LIN {X 0,Y 298.413,Z 394.313,A -85,B 0,C 180,E1 -16229.642,E2 -16229.642} C_VEL
LIN {X 0,Y 298.389,Z 394.317,A -85,B 0,C 180,E1 -16232.801,E2 -16232.801} C_VEL
LIN {X 0,Y 298.456,Z 394.307,A -85,B 0,C 180,E1 -16236.814,E2 -16236.814} C_VEL
LIN {X 0,Y 298.404,Z 394.314,A -85,B 0,C 180,E1 -16241.095,E2 -16241.095} C_VEL
LIN {X 0,Y 298.418,Z 394.313,A -85,B 0,C 180,E1 -16243.11,E2 -16243.11} C_VEL
LIN {X 0,Y 298.396,Z 394.317,A -85,B 0,C 180,E1 -16246.922,E2 -16246.922} C_VEL
LIN {X 0,Y 298.398,Z 394.314,A -85,B 0,C 180,E1 -16251.008,E2 -16251.008} C_VEL
LIN {X 0,Y 298.421,Z 394.313,A -85,B 0,C 180,E1 -16254.764,E2 -16254.764} C_VEL
LIN {X 0,Y 298.43,Z 394.322,A -85,B 0,C 180,E1 -16255.234,E2 -16255.234} C_VEL
LIN {X 0,Y 298.861,Z 396.048,A -85,B 0,C 180,E1 -16255.643,E2 -16255.643} C_VEL
LIN {X 0,Y 302.324,Z 402.19,A -85,B 0,C 180,E1 -16257.395,E2 -16257.395} C_VEL
LIN {X 0,Y 303.861,Z 406.66,A -85,B 0,C 180,E1 -16258.271,E2 -16258.271} C_VEL
LIN {X 0,Y 306.901,Z 413.206,A -85,B 0,C 180,E1 -16259.176,E2 -16259.176} C_VEL
LIN {X 0,Y 310.226,Z 420.843,A -85,B 0,C 180,E1 -16260.12,E2 -16260.12} C_VEL
LIN {X 0,Y 313.351,Z 428.982,A -85,B 0,C 180,E1 -16261.011,E2 -16261.011} C_VEL
LIN {X 0,Y 315.702,Z 443.344,A -85,B 0,C 180,E1 -16261.99,E2 -16261.99} C_VEL
LIN {X 0,Y 317.187,Z 456.396,A -85,B 0,C 180,E1 -16262.756,E2 -16262.756} C_VEL
LIN {X 0,Y 317.42,Z 461.154,A -85,B 0,C 180,E1 -16262.981,E2 -16262.981} C_VEL
LIN {X 0,Y 313.679,Z 525.311,A -85,B 0,C 180,E1 -16265.029,E2 -16265.029} C_VEL
LIN {X 0,Y 312.276,Z 538.46,A -85,B 0,C 180,E1 -16265.663,E2 -16265.663} C_VEL
LIN {X 0,Y 310.663,Z 550.678,A -85,B 0,C 180,E1 -16266.504,E2 -16266.504} C_VEL
LIN {X 0,Y 308.807,Z 562.616,A -85,B 0,C 180,E1 -16267.594,E2 -16267.594} C_VEL
LIN {X 0,Y 306.824,Z 573.531,A -85,B 0,C 180,E1 -16268.855,E2 -16268.855} C_VEL
LIN {X 0,Y 304.681,Z 584.454,A -85,B 0,C 180,E1 -16270.462,E2 -16270.462} C_VEL
LIN {X 0,Y 302.875,Z 593.194,A -85,B 0,C 180,E1 -16272.06,E2 -16272.06} C_VEL
LIN {X 0,Y 301.068,Z 602.117,A -85,B 0,C 180,E1 -16274.082,E2 -16274.082} C_VEL
LIN {X 0,Y 299.516,Z 609.166,A -85,B 0,C 180,E1 -16276.085,E2 -16276.085} C_VEL
LIN {X 0,Y 298.089,Z 615.668,A -85,B 0,C 180,E1 -16278.441,E2 -16278.441} C_VEL
LIN {X 0,Y 297.32,Z 619.91,A -85,B 0,C 180,E1 -16280.478,E2 -16280.478} C_VEL
LIN {X 0,Y 296.96,Z 622.117,A -85,B 0,C 180,E1 -16281.838,E2 -16281.838} C_VEL
LIN {X 0,Y 296.586,Z 625.088,A -85,B 0,C 180,E1 -16284.412,E2 -16284.412} C_VEL
LIN {X 0,Y 296.494,Z 627.829,A -85,B 0,C 180,E1 -16288.644,E2 -16288.644} C_VEL
LIN {X 0,Y 296.518,Z 628.283,A -85,B 0,C 180,E1 -16290.002,E2 -16290.002} C_VEL
LIN {X 0,Y 296.485,Z 628.313,A -85,B 0,C 180,E1 -16291.36,E2 -16291.36} C_VEL
LIN {X 0,Y 296.527,Z 627.952,A -85,B 0,C 180,E1 -16292.719,E2 -16292.719} C_VEL
LIN {X 0,Y 296.493,Z 627.197,A -85,B 0,C 180,E1 -16294.08,E2 -16294.08} C_VEL
LIN {X 0,Y 296.547,Z 625.934,A -85,B 0,C 180,E1 -16295.51,E2 -16295.51} C_VEL
LIN {X 0,Y 296.948,Z 622.356,A -85,B 0,C 180,E1 -16298.166,E2 -16298.166} C_VEL
LIN {X 0,Y 297.479,Z 618.423,A -85,B 0,C 180,E1 -16300.208,E2 -16300.208} C_VEL
LIN {X 0,Y 298.337,Z 613.363,A -85,B 0,C 180,E1 -16302.242,E2 -16302.242} C_VEL
LIN {X 0,Y 299.641,Z 607.023,A -85,B 0,C 180,E1 -16304.259,E2 -16304.259} C_VEL
LIN {X 0,Y 301.128,Z 599.116,A -85,B 0,C 180,E1 -16306.266,E2 -16306.266} C_VEL
LIN {X 0,Y 302.907,Z 589.288,A -85,B 0,C 180,E1 -16308.255,E2 -16308.255} C_VEL
LIN {X 0,Y 304.715,Z 579.147,A -85,B 0,C 180,E1 -16309.89,E2 -16309.89} C_VEL
LIN {X 0,Y 306.713,Z 567.717,A -85,B 0,C 180,E1 -16311.333,E2 -16311.333} C_VEL
LIN {X 0,Y 308.342,Z 556.565,A -85,B 0,C 180,E1 -16312.446,E2 -16312.446} C_VEL
LIN {X 0,Y 309.823,Z 544.144,A -85,B 0,C 180,E1 -16313.39,E2 -16313.39} C_VEL
LIN {X 0,Y 311.118,Z 531.155,A -85,B 0,C 180,E1 -16314.08,E2 -16314.08} C_VEL
LIN {X 0,Y 311.871,Z 518.085,A -85,B 0,C 180,E1 -16314.534,E2 -16314.534} C_VEL
LIN {X 0,Y 313.809,Z 459.058,A -85,B 0,C 180,E1 -16316.022,E2 -16316.022} C_VEL
LIN {X 0,Y 310.871,Z 439.691,A -85,B 0,C 180,E1 -16316.91,E2 -16316.91} C_VEL
LIN {X 0,Y 308.062,Z 426.174,A -85,B 0,C 180,E1 -16317.642,E2 -16317.642} C_VEL
LIN {X 0,Y 303.315,Z 415.098,A -85,B 0,C 180,E1 -16318.585,E2 -16318.585} C_VEL
LIN {X 0,Y 301.215,Z 405.403,A -85,B 0,C 180,E1 -16322.062,E2 -16322.062} C_VEL
LIN {X 0,Y 299.211,Z 397.209,A -85,B 0,C 180,E1 -16325.239,E2 -16325.239} C_VEL
LIN {X 0,Y 298.473,Z 394.309,A -85,B 0,C 180,E1 -16326.437,E2 -16326.437} C_VEL
LIN {X 0,Y 298.414,Z 394.321,A -85,B 0,C 180,E1 -16329.487,E2 -16329.487} C_VEL
LIN {X 0,Y 298.404,Z 394.318,A -85,B 0,C 180,E1 -16333.104,E2 -16333.104} C_VEL
LIN {X 0,Y 298.408,Z 394.312,A -85,B 0,C 180,E1 -16336.922,E2 -16336.922} C_VEL
LIN {X 0,Y 298.41,Z 394.314,A -85,B 0,C 180,E1 -16341.007,E2 -16341.007} C_VEL
LIN {X 0,Y 298.425,Z 394.31,A -85,B 0,C 180,E1 -16343.931,E2 -16343.931} C_VEL
LIN {X 0,Y 298.4,Z 394.314,A -85,B 0,C 180,E1 -16347.985,E2 -16347.985} C_VEL
LIN {X 0,Y 298.463,Z 394.306,A -85,B 0,C 180,E1 -16351.904,E2 -16351.904} C_VEL
LIN {X 0,Y 298.49,Z 394.305,A -85,B 0,C 180,E1 -16354.924,E2 -16354.924} C_VEL
LIN {X 0,Y 298.457,Z 394.308,A -85,B 0,C 180,E1 -16359.316,E2 -16359.316} C_VEL
LIN {X 0,Y 298.545,Z 394.289,A -85,B 0,C 180,E1 -16362.18,E2 -16362.18} C_VEL
LIN {X 0,Y 298.6,Z 394.28,A -85,B 0,C 180,E1 -16364.995,E2 -16364.995} C_VEL
LIN {X 0,Y 298.6,Z 394.28,A -85,B 0,C 180,E1 -16369.147,E2 -16369.147} C_VEL
LIN {X 0,Y 298.766,Z 394.271,A -85,B 0,C 180,E1 -16371.886,E2 -16371.886} C_VEL
LIN {X 0,Y 298.667,Z 394.28,A -85,B 0,C 180,E1 -16374.599,E2 -16374.599} C_VEL
LIN {X 0,Y 298.929,Z 394.25,A -85,B 0,C 180,E1 -16378.653,E2 -16378.653} C_VEL
LIN {X 0,Y 298.929,Z 394.245,A -85,B 0,C 180,E1 -16381.347,E2 -16381.347} C_VEL
LIN {X 0,Y 298.805,Z 394.26,A -85,B 0,C 180,E1 -16386.754,E2 -16386.754} C_VEL
LIN {X 0,Y 298.688,Z 394.277,A -85,B 0,C 180,E1 -16389.48,E2 -16389.48} C_VEL
LIN {X 0,Y 298.559,Z 394.295,A -85,B 0,C 180,E1 -16393.615,E2 -16393.615} C_VEL
LIN {X 0,Y 298.556,Z 394.296,A -85,B 0,C 180,E1 -16396.408,E2 -16396.408} C_VEL
LIN {X 0,Y 298.556,Z 394.478,A -85,B 0,C 180,E1 -16399.762,E2 -16399.762} C_VEL
LIN {X 0,Y 300.424,Z 402.299,A -85,B 0,C 180,E1 -16403.115,E2 -16403.115} C_VEL
LIN {X 0,Y 308.076,Z 417.875,A -85,B 0,C 180,E1 -16404.576,E2 -16404.576} C_VEL
LIN {X 0,Y 313.726,Z 431.385,A -85,B 0,C 180,E1 -16405.635,E2 -16405.635} C_VEL
LIN {X 0,Y 314.519,Z 435.202,A -85,B 0,C 180,E1 -16405.832,E2 -16405.832} C_VEL
LIN {X 0,Y 311.916,Z 509.359,A -85,B 0,C 180,E1 -16407.731,E2 -16407.731} C_VEL
LIN {X 0,Y 311.021,Z 522.182,A -85,B 0,C 180,E1 -16408.298,E2 -16408.298} C_VEL
LIN {X 0,Y 309.823,Z 534.58,A -85,B 0,C 180,E1 -16409.097,E2 -16409.097} C_VEL
LIN {X 0,Y 308.255,Z 547.18,A -85,B 0,C 180,E1 -16410.211,E2 -16410.211} C_VEL
LIN {X 0,Y 306.574,Z 558.665,A -85,B 0,C 180,E1 -16411.537,E2 -16411.537} C_VEL
LIN {X 0,Y 304.885,Z 568.72,A -85,B 0,C 180,E1 -16412.997,E2 -16412.997} C_VEL
LIN {X 0,Y 303.175,Z 577.721,A -85,B 0,C 180,E1 -16414.618,E2 -16414.618} C_VEL
LIN {X 0,Y 301.474,Z 586.009,A -85,B 0,C 180,E1 -16416.458,E2 -16416.458} C_VEL
LIN {X 0,Y 300.068,Z 592.824,A -85,B 0,C 180,E1 -16418.328,E2 -16418.328} C_VEL
LIN {X 0,Y 298.765,Z 599.542,A -85,B 0,C 180,E1 -16420.671,E2 -16420.671} C_VEL
LIN {X 0,Y 297.704,Z 604.913,A -85,B 0,C 180,E1 -16423.206,E2 -16423.206} C_VEL
LIN {X 0,Y 297.085,Z 607.992,A -85,B 0,C 180,E1 -16425.211,E2 -16425.211} C_VEL
LIN {X 0,Y 296.595,Z 610.168,A -85,B 0,C 180,E1 -16427.271,E2 -16427.271} C_VEL
LIN {X 0,Y 296.321,Z 611.406,A -85,B 0,C 180,E1 -16429.373,E2 -16429.373} C_VEL
LIN {X 0,Y 296.196,Z 611.621,A -85,B 0,C 180,E1 -16431.907,E2 -16431.907} C_VEL
LIN {X 0,Y 296.212,Z 610.875,A -85,B 0,C 180,E1 -16433.775,E2 -16433.775} C_VEL
LIN {X 0,Y 296.464,Z 608.905,A -85,B 0,C 180,E1 -16436.07,E2 -16436.07} C_VEL
LIN {X 0,Y 296.925,Z 605.306,A -85,B 0,C 180,E1 -16438.617,E2 -16438.617} C_VEL
LIN {X 0,Y 297.467,Z 600.516,A -85,B 0,C 180,E1 -16440.947,E2 -16440.947} C_VEL
LIN {X 0,Y 298.229,Z 594.935,A -85,B 0,C 180,E1 -16443.021,E2 -16443.021} C_VEL
LIN {X 0,Y 299.112,Z 588.328,A -85,B 0,C 180,E1 -16444.979,E2 -16444.979} C_VEL
LIN {X 0,Y 300.263,Z 580.217,A -85,B 0,C 180,E1 -16446.916,E2 -16446.916} C_VEL
LIN {X 0,Y 301.61,Z 570.524,A -85,B 0,C 180,E1 -16448.76,E2 -16448.76} C_VEL
LIN {X 0,Y 303.001,Z 560.131,A -85,B 0,C 180,E1 -16450.345,E2 -16450.345} C_VEL
LIN {X 0,Y 304.294,Z 549.028,A -85,B 0,C 180,E1 -16451.697,E2 -16451.697} C_VEL
LIN {X 0,Y 305.496,Z 536.723,A -85,B 0,C 180,E1 -16452.856,E2 -16452.856} C_VEL
LIN {X 0,Y 306.524,Z 523.684,A -85,B 0,C 180,E1 -16453.772,E2 -16453.772} C_VEL
LIN {X 0,Y 307.343,Z 510.203,A -85,B 0,C 180,E1 -16454.405,E2 -16454.405} C_VEL
LIN {X 0,Y 308.068,Z 485.661,A -85,B 0,C 180,E1 -16455.068,E2 -16455.068} C_VEL
LIN {X 0,Y 309.548,Z 432.634,A -85,B 0,C 180,E1 -16456.374,E2 -16456.374} C_VEL
LIN {X 0,Y 307.146,Z 421.12,A -85,B 0,C 180,E1 -16456.855,E2 -16456.855} C_VEL
LIN {X 0,Y 299.859,Z 400.774,A -85,B 0,C 180,E1 -16457.993,E2 -16457.993} C_VEL
LIN {X 0,Y 298.652,Z 394.286,A -85,B 0,C 180,E1 -16460.346,E2 -16460.346} C_VEL
LIN {X 0,Y 298.75,Z 394.27,A -85,B 0,C 180,E1 -16463.243,E2 -16463.243} C_VEL
LIN {X 0,Y 298.839,Z 394.259,A -85,B 0,C 180,E1 -16467.302,E2 -16467.302} C_VEL
LIN {X 0,Y 299.012,Z 394.239,A -85,B 0,C 180,E1 -16469.998,E2 -16469.998} C_VEL
LIN {X 0,Y 298.84,Z 394.258,A -85,B 0,C 180,E1 -16472.694,E2 -16472.694} C_VEL
LIN {X 0,Y 298.8,Z 394.262,A -85,B 0,C 180,E1 -16476.752,E2 -16476.752} C_VEL
LIN {X 0,Y 298.682,Z 394.278,A -85,B 0,C 180,E1 -16479.479,E2 -16479.479} C_VEL
LIN {X 0,Y 298.553,Z 394.293,A -85,B 0,C 180,E1 -16483.613,E2 -16483.613} C_VEL
LIN {X 0,Y 298.549,Z 394.296,A -85,B 0,C 180,E1 -16486.407,E2 -16486.407} C_VEL
LIN {X 0,Y 298.509,Z 394.298,A -85,B 0,C 180,E1 -16489.652,E2 -16489.652} C_VEL
LIN {X 0,Y 298.453,Z 394.309,A -85,B 0,C 180,E1 -16493.596,E2 -16493.596} C_VEL
LIN {X 0,Y 298.487,Z 394.298,A -85,B 0,C 180,E1 -16496.572,E2 -16496.572} C_VEL
LIN {X 0,Y 298.419,Z 394.31,A -85,B 0,C 180,E1 -16499.639,E2 -16499.639} C_VEL
LIN {X 0,Y 298.394,Z 394.313,A -85,B 0,C 180,E1 -16502.798,E2 -16502.798} C_VEL
LIN {X 0,Y 298.466,Z 394.304,A -85,B 0,C 180,E1 -16506.812,E2 -16506.812} C_VEL
LIN {X 0,Y 298.413,Z 394.312,A -85,B 0,C 180,E1 -16511.093,E2 -16511.093} C_VEL
LIN {X 0,Y 298.485,Z 394.46,A -85,B 0,C 180,E1 -16512.259,E2 -16512.259} C_VEL
LIN {X 0,Y 299.327,Z 398.591,A -85,B 0,C 180,E1 -16513.333,E2 -16513.333} C_VEL
LIN {X 0,Y 304.933,Z 417.141,A -85,B 0,C 180,E1 -16514.243,E2 -16514.243} C_VEL
LIN {X 0,Y 307.315,Z 432.432,A -85,B 0,C 180,E1 -16514.851,E2 -16514.851} C_VEL
LIN {X 0,Y 306.451,Z 459.715,A -85,B 0,C 180,E1 -16515.644,E2 -16515.644} C_VEL
LIN {X 0,Y 305.703,Z 465.514,A -85,B 0,C 180,E1 -16515.784,E2 -16515.784} C_VEL
LIN {X 0,Y 299.506,Z 484.299,A -85,B 0,C 180,E1 -16516.06,E2 -16516.06} C_VEL
LIN {X 0,Y 298.583,Z 490.102,A -85,B 0,C 180,E1 -16516.198,E2 -16516.198} C_VEL
LIN {X 0,Y 297.795,Z 511.029,A -85,B 0,C 180,E1 -16516.881,E2 -16516.881} C_VEL
LIN {X 0,Y 297.105,Z 524.525,A -85,B 0,C 180,E1 -16517.61,E2 -16517.61} C_VEL
LIN {X 0,Y 296.156,Z 537.069,A -85,B 0,C 180,E1 -16518.552,E2 -16518.552} C_VEL
LIN {X 0,Y 295.041,Z 549.89,A -85,B 0,C 180,E1 -16519.839,E2 -16519.839} C_VEL
LIN {X 0,Y 294.041,Z 560.159,A -85,B 0,C 180,E1 -16521.14,E2 -16521.14} C_VEL
LIN {X 0,Y 292.912,Z 570.755,A -85,B 0,C 180,E1 -16522.814,E2 -16522.814} C_VEL
LIN {X 0,Y 291.816,Z 580.381,A -85,B 0,C 180,E1 -16524.689,E2 -16524.689} C_VEL
LIN {X 0,Y 290.987,Z 588.658,A -85,B 0,C 180,E1 -16526.711,E2 -16526.711} C_VEL
LIN {X 0,Y 290.264,Z 596.232,A -85,B 0,C 180,E1 -16529.035,E2 -16529.035} C_VEL
LIN {X 0,Y 289.826,Z 601.225,A -85,B 0,C 180,E1 -16530.989,E2 -16530.989} C_VEL
LIN {X 0,Y 289.473,Z 605.746,A -85,B 0,C 180,E1 -16533.311,E2 -16533.311} C_VEL
LIN {X 0,Y 289.163,Z 608.885,A -85,B 0,C 180,E1 -16535.595,E2 -16535.595} C_VEL
LIN {X 0,Y 289.088,Z 610.571,A -85,B 0,C 180,E1 -16537.485,E2 -16537.485} C_VEL
LIN {X 0,Y 289.225,Z 611.599,A -85,B 0,C 180,E1 -16540.111,E2 -16540.111} C_VEL
LIN {X 0,Y 289.438,Z 611.526,A -85,B 0,C 180,E1 -16541.599,E2 -16541.599} C_VEL
LIN {X 0,Y 289.627,Z 610.951,A -85,B 0,C 180,E1 -16543.071,E2 -16543.071} C_VEL
LIN {X 0,Y 290.264,Z 608.927,A -85,B 0,C 180,E1 -16545.571,E2 -16545.571} C_VEL
LIN {X 0,Y 291.274,Z 605.287,A -85,B 0,C 180,E1 -16548.165,E2 -16548.165} C_VEL
LIN {X 0,Y 292.433,Z 600.999,A -85,B 0,C 180,E1 -16550.315,E2 -16550.315} C_VEL
LIN {X 0,Y 293.933,Z 595.453,A -85,B 0,C 180,E1 -16552.443,E2 -16552.443} C_VEL
LIN {X 0,Y 295.713,Z 588.491,A -85,B 0,C 180,E1 -16554.545,E2 -16554.545} C_VEL
LIN {X 0,Y 297.866,Z 579.71,A -85,B 0,C 180,E1 -16556.618,E2 -16556.618} C_VEL
LIN {X 0,Y 299.917,Z 570.738,A -85,B 0,C 180,E1 -16558.321,E2 -16558.321} C_VEL
LIN {X 0,Y 302.247,Z 559.672,A -85,B 0,C 180,E1 -16560,E2 -16560} C_VEL
LIN {X 0,Y 304.293,Z 548.681,A -85,B 0,C 180,E1 -16561.323,E2 -16561.323} C_VEL
LIN {X 0,Y 306.132,Z 536.555,A -85,B 0,C 180,E1 -16562.467,E2 -16562.467} C_VEL
LIN {X 0,Y 307.812,Z 522.802,A -85,B 0,C 180,E1 -16563.436,E2 -16563.436} C_VEL
LIN {X 0,Y 309.15,Z 508.158,A -85,B 0,C 180,E1 -16564.12,E2 -16564.12} C_VEL
LIN {X 0,Y 313.602,Z 438.511,A -85,B 0,C 180,E1 -16566.341,E2 -16566.341} C_VEL
LIN {X 0,Y 311.585,Z 432.983,A -85,B 0,C 180,E1 -16566.903,E2 -16566.903} C_VEL
LIN {X 0,Y 304.494,Z 418.301,A -85,B 0,C 180,E1 -16568.83,E2 -16568.83} C_VEL
LIN {X 0,Y 299.451,Z 409.843,A -85,B 0,C 180,E1 -16570.265,E2 -16570.265} C_VEL
LIN {X 0,Y 295.899,Z 404.495,A -85,B 0,C 180,E1 -16571.322,E2 -16571.322} C_VEL
LIN {X 0,Y 293.577,Z 400.956,A -85,B 0,C 180,E1 -16572.091,E2 -16572.091} C_VEL
LIN {X 0,Y 292.706,Z 398.323,A -85,B 0,C 180,E1 -16573.185,E2 -16573.185} C_VEL
LIN {X 0,Y 291.554,Z 395.399,A -85,B 0,C 180,E1 -16574.483,E2 -16574.483} C_VEL
LIN {X 0,Y 291.531,Z 395.174,A -85,B 0,C 180,E1 -16574.662,E2 -16574.662} C_VEL
LIN {X 0,Y 291.476,Z 395.178,A -85,B 0,C 180,E1 -16578.267,E2 -16578.267} C_VEL
LIN {X 0,Y 291.411,Z 395.185,A -85,B 0,C 180,E1 -16581.208,E2 -16581.208} C_VEL
LIN {X 0,Y 291.428,Z 395.183,A -85,B 0,C 180,E1 -16584.203,E2 -16584.203} C_VEL
LIN {X 0,Y 291.414,Z 395.187,A -85,B 0,C 180,E1 -16587.272,E2 -16587.272} C_VEL
LIN {X 0,Y 291.331,Z 395.197,A -85,B 0,C 180,E1 -16590.438,E2 -16590.438} C_VEL
LIN {X 0,Y 291.337,Z 395.193,A -85,B 0,C 180,E1 -16593.699,E2 -16593.699} C_VEL
LIN {X 0,Y 291.386,Z 395.187,A -85,B 0,C 180,E1 -16597.26,E2 -16597.26} C_VEL
LIN {X 0,Y 291.363,Z 395.19,A -85,B 0,C 180,E1 -16600.637,E2 -16600.637} C_VEL
LIN {X 0,Y 291.315,Z 395.195,A -85,B 0,C 180,E1 -16604.397,E2 -16604.397} C_VEL
LIN {X 0,Y 291.321,Z 395.197,A -85,B 0,C 180,E1 -16608.406,E2 -16608.406} C_VEL
LIN {X 0,Y 291.347,Z 395.193,A -85,B 0,C 180,E1 -16611.16,E2 -16611.16} C_VEL
LIN {X 0,Y 291.397,Z 395.254,A -85,B 0,C 180,E1 -16613.525,E2 -16613.525} C_VEL
LIN {X 0,Y 292.249,Z 397.821,A -85,B 0,C 180,E1 -16614.272,E2 -16614.272} C_VEL
LIN {X 0,Y 293.609,Z 399.559,A -85,B 0,C 180,E1 -16614.939,E2 -16614.939} C_VEL
LIN {X 0,Y 297.061,Z 406.347,A -85,B 0,C 180,E1 -16616.824,E2 -16616.824} C_VEL
LIN {X 0,Y 299.504,Z 411,A -85,B 0,C 180,E1 -16617.6,E2 -16617.6} C_VEL
LIN {X 0,Y 303.218,Z 419.259,A -85,B 0,C 180,E1 -16618.764,E2 -16618.764} C_VEL
LIN {X 0,Y 307.157,Z 428.909,A -85,B 0,C 180,E1 -16619.949,E2 -16619.949} C_VEL
LIN {X 0,Y 308.561,Z 433.561,A -85,B 0,C 180,E1 -16620.41,E2 -16620.41} C_VEL
LIN {X 0,Y 310.991,Z 450.796,A -85,B 0,C 180,E1 -16621.579,E2 -16621.579} C_VEL
LIN {X 0,Y 311.898,Z 461.029,A -85,B 0,C 180,E1 -16622.158,E2 -16622.158} C_VEL
LIN {X 0,Y 307.844,Z 525.772,A -85,B 0,C 180,E1 -16624.295,E2 -16624.295} C_VEL
LIN {X 0,Y 306.308,Z 539.366,A -85,B 0,C 180,E1 -16624.976,E2 -16624.976} C_VEL
LIN {X 0,Y 304.605,Z 551.25,A -85,B 0,C 180,E1 -16625.826,E2 -16625.826} C_VEL
LIN {X 0,Y 302.364,Z 564.475,A -85,B 0,C 180,E1 -16627.089,E2 -16627.089} C_VEL
LIN {X 0,Y 300.087,Z 576.022,A -85,B 0,C 180,E1 -16628.537,E2 -16628.537} C_VEL
LIN {X 0,Y 298.073,Z 585.483,A -85,B 0,C 180,E1 -16630.01,E2 -16630.01} C_VEL
LIN {X 0,Y 296.179,Z 594.087,A -85,B 0,C 180,E1 -16631.651,E2 -16631.651} C_VEL
LIN {X 0,Y 294.538,Z 601.432,A -85,B 0,C 180,E1 -16633.363,E2 -16633.363} C_VEL
LIN {X 0,Y 292.868,Z 608.544,A -85,B 0,C 180,E1 -16635.408,E2 -16635.408} C_VEL
LIN {X 0,Y 291.468,Z 614.275,A -85,B 0,C 180,E1 -16637.468,E2 -16637.468} C_VEL
LIN {X 0,Y 290.53,Z 618.788,A -85,B 0,C 180,E1 -16639.549,E2 -16639.549} C_VEL
LIN {X 0,Y 289.91,Z 622.193,A -85,B 0,C 180,E1 -16641.638,E2 -16641.638} C_VEL
LIN {X 0,Y 289.669,Z 623.899,A -85,B 0,C 180,E1 -16643.034,E2 -16643.034} C_VEL
LIN {X 0,Y 289.516,Z 625.177,A -85,B 0,C 180,E1 -16644.43,E2 -16644.43} C_VEL
LIN {X 0,Y 289.459,Z 626.662,A -85,B 0,C 180,E1 -16647.218,E2 -16647.218} C_VEL
LIN {X 0,Y 289.416,Z 627.573,A -85,B 0,C 180,E1 -16648.61,E2 -16648.61} C_VEL
LIN {X 0,Y 289.436,Z 628.069,A -85,B 0,C 180,E1 -16650.002,E2 -16650.002} C_VEL
LIN {X 0,Y 289.407,Z 628.122,A -85,B 0,C 180,E1 -16651.393,E2 -16651.393} C_VEL
LIN {X 0,Y 289.43,Z 627.781,A -85,B 0,C 180,E1 -16652.785,E2 -16652.785} C_VEL
LIN {X 0,Y 289.428,Z 626.074,A -85,B 0,C 180,E1 -16655.39,E2 -16655.39} C_VEL
LIN {X 0,Y 289.733,Z 623.374,A -85,B 0,C 180,E1 -16657.669,E2 -16657.669} C_VEL
LIN {X 0,Y 290.263,Z 619.838,A -85,B 0,C 180,E1 -16659.76,E2 -16659.76} C_VEL
LIN {X 0,Y 291.087,Z 615.214,A -85,B 0,C 180,E1 -16661.844,E2 -16661.844} C_VEL
LIN {X 0,Y 292.505,Z 608.242,A -85,B 0,C 180,E1 -16664.259,E2 -16664.259} C_VEL
LIN {X 0,Y 294.066,Z 600.724,A -85,B 0,C 180,E1 -16666.311,E2 -16666.311} C_VEL
LIN {X 0,Y 295.502,Z 593.087,A -85,B 0,C 180,E1 -16668.012,E2 -16668.012} C_VEL
LIN {X 0,Y 297.312,Z 583.863,A -85,B 0,C 180,E1 -16669.687,E2 -16669.687} C_VEL
LIN {X 0,Y 299.198,Z 573.641,A -85,B 0,C 180,E1 -16671.173,E2 -16671.173} C_VEL
LIN {X 0,Y 301.105,Z 562.366,A -85,B 0,C 180,E1 -16672.472,E2 -16672.472} C_VEL
LIN {X 0,Y 302.692,Z 550.765,A -85,B 0,C 180,E1 -16673.521,E2 -16673.521} C_VEL
LIN {X 0,Y 304.151,Z 538.255,A -85,B 0,C 180,E1 -16674.352,E2 -16674.352} C_VEL
LIN {X 0,Y 305.381,Z 524.258,A -85,B 0,C 180,E1 -16674.973,E2 -16674.973} C_VEL
LIN {X 0,Y 307.617,Z 459.696,A -85,B 0,C 180,E1 -16676.682,E2 -16676.682} C_VEL
LIN {X 0,Y 304.895,Z 441.36,A -85,B 0,C 180,E1 -16677.557,E2 -16677.557} C_VEL
LIN {X 0,Y 302.324,Z 428.984,A -85,B 0,C 180,E1 -16678.251,E2 -16678.251} C_VEL
LIN {X 0,Y 297.367,Z 417.87,A -85,B 0,C 180,E1 -16679.242,E2 -16679.242} C_VEL
LIN {X 0,Y 296.14,Z 414.849,A -85,B 0,C 180,E1 -16679.526,E2 -16679.526} C_VEL
LIN {X 0,Y 293.791,Z 404.639,A -85,B 0,C 180,E1 -16683.383,E2 -16683.383} C_VEL
LIN {X 0,Y 291.844,Z 396.857,A -85,B 0,C 180,E1 -16686.586,E2 -16686.586} C_VEL
LIN {X 0,Y 291.406,Z 395.19,A -85,B 0,C 180,E1 -16687.354,E2 -16687.354} C_VEL
LIN {X 0,Y 291.34,Z 395.198,A -85,B 0,C 180,E1 -16690.643,E2 -16690.643} C_VEL
LIN {X 0,Y 291.296,Z 395.2,A -85,B 0,C 180,E1 -16694.403,E2 -16694.403} C_VEL
LIN {X 0,Y 291.333,Z 395.196,A -85,B 0,C 180,E1 -16698.405,E2 -16698.405} C_VEL
LIN {X 0,Y 291.359,Z 395.194,A -85,B 0,C 180,E1 -16701.159,E2 -16701.159} C_VEL
LIN {X 0,Y 291.367,Z 395.193,A -85,B 0,C 180,E1 -16704.627,E2 -16704.627} C_VEL
LIN {X 0,Y 291.377,Z 395.189,A -85,B 0,C 180,E1 -16707.951,E2 -16707.951} C_VEL
LIN {X 0,Y 291.384,Z 395.189,A -85,B 0,C 180,E1 -16711.159,E2 -16711.159} C_VEL
LIN {X 0,Y 291.419,Z 395.178,A -85,B 0,C 180,E1 -16714.272,E2 -16714.272} C_VEL
LIN {X 0,Y 291.388,Z 395.178,A -85,B 0,C 180,E1 -16717.3,E2 -16717.3} C_VEL
LIN {X 0,Y 291.465,Z 395.174,A -85,B 0,C 180,E1 -16720.271,E2 -16720.271} C_VEL
LIN {X 0,Y 291.562,Z 395.159,A -85,B 0,C 180,E1 -16724.624,E2 -16724.624} C_VEL
LIN {X 0,Y 291.544,Z 395.16,A -85,B 0,C 180,E1 -16728.881,E2 -16728.881} C_VEL
LIN {X 0,Y 291.717,Z 395.148,A -85,B 0,C 180,E1 -16731.689,E2 -16731.689} C_VEL
LIN {X 0,Y 291.637,Z 395.154,A -85,B 0,C 180,E1 -16734.469,E2 -16734.469} C_VEL
LIN {X 0,Y 291.895,Z 395.126,A -85,B 0,C 180,E1 -16738.62,E2 -16738.62} C_VEL
LIN {X 0,Y 291.895,Z 395.122,A -85,B 0,C 180,E1 -16741.38,E2 -16741.38} C_VEL
LIN {X 0,Y 291.754,Z 395.138,A -85,B 0,C 180,E1 -16746.918,E2 -16746.918} C_VEL
LIN {X 0,Y 291.637,Z 395.155,A -85,B 0,C 180,E1 -16749.712,E2 -16749.712} C_VEL
LIN {X 0,Y 291.529,Z 395.169,A -85,B 0,C 180,E1 -16753.95,E2 -16753.95} C_VEL
LIN {X 0,Y 291.495,Z 395.178,A -85,B 0,C 180,E1 -16756.818,E2 -16756.818} C_VEL
LIN {X 0,Y 291.532,Z 395.353,A -85,B 0,C 180,E1 -16758.902,E2 -16758.902} C_VEL
LIN {X 0,Y 293.317,Z 402.744,A -85,B 0,C 180,E1 -16762.172,E2 -16762.172} C_VEL
LIN {X 0,Y 301.287,Z 418.495,A -85,B 0,C 180,E1 -16763.761,E2 -16763.761} C_VEL
LIN {X 0,Y 306.31,Z 429.899,A -85,B 0,C 180,E1 -16764.731,E2 -16764.731} C_VEL
LIN {X 0,Y 308.228,Z 435.316,A -85,B 0,C 180,E1 -16765.122,E2 -16765.122} C_VEL
LIN {X 0,Y 308.419,Z 438.295,A -85,B 0,C 180,E1 -16765.234,E2 -16765.234} C_VEL
LIN {X 0,Y 305.723,Z 509.386,A -85,B 0,C 180,E1 -16767.094,E2 -16767.094} C_VEL
LIN {X 0,Y 304.773,Z 522.165,A -85,B 0,C 180,E1 -16767.663,E2 -16767.663} C_VEL
LIN {X 0,Y 303.545,Z 534.583,A -85,B 0,C 180,E1 -16768.475,E2 -16768.475} C_VEL
LIN {X 0,Y 302.118,Z 545.852,A -85,B 0,C 180,E1 -16769.464,E2 -16769.464} C_VEL
LIN {X 0,Y 300.355,Z 557.445,A -85,B 0,C 180,E1 -16770.788,E2 -16770.788} C_VEL
LIN {X 0,Y 298.707,Z 566.742,A -85,B 0,C 180,E1 -16772.11,E2 -16772.11} C_VEL
LIN {X 0,Y 296.979,Z 575.886,A -85,B 0,C 180,E1 -16773.708,E2 -16773.708} C_VEL
LIN {X 0,Y 295.101,Z 584.618,A -85,B 0,C 180,E1 -16775.586,E2 -16775.586} C_VEL
LIN {X 0,Y 293.355,Z 592.558,A -85,B 0,C 180,E1 -16777.757,E2 -16777.757} C_VEL
LIN {X 0,Y 292.214,Z 598.143,A -85,B 0,C 180,E1 -16779.677,E2 -16779.677} C_VEL
LIN {X 0,Y 291.252,Z 602.591,A -85,B 0,C 180,E1 -16781.577,E2 -16781.577} C_VEL
LIN {X 0,Y 290.521,Z 606.088,A -85,B 0,C 180,E1 -16783.468,E2 -16783.468} C_VEL
LIN {X 0,Y 289.95,Z 608.687,A -85,B 0,C 180,E1 -16785.336,E2 -16785.336} C_VEL
LIN {X 0,Y 289.53,Z 610.467,A -85,B 0,C 180,E1 -16787.18,E2 -16787.18} C_VEL
LIN {X 0,Y 289.276,Z 611.543,A -85,B 0,C 180,E1 -16789.005,E2 -16789.005} C_VEL
LIN {X 0,Y 289.114,Z 611.927,A -85,B 0,C 180,E1 -16791.067,E2 -16791.067} C_VEL
LIN {X 0,Y 289.096,Z 611.306,A -85,B 0,C 180,E1 -16793.345,E2 -16793.345} C_VEL
LIN {X 0,Y 289.383,Z 609.143,A -85,B 0,C 180,E1 -16796.04,E2 -16796.04} C_VEL
LIN {X 0,Y 289.724,Z 606.419,A -85,B 0,C 180,E1 -16798.105,E2 -16798.105} C_VEL
LIN {X 0,Y 290.301,Z 601.701,A -85,B 0,C 180,E1 -16800.638,E2 -16800.638} C_VEL
LIN {X 0,Y 290.973,Z 596.624,A -85,B 0,C 180,E1 -16802.681,E2 -16802.681} C_VEL
LIN {X 0,Y 291.884,Z 590.321,A -85,B 0,C 180,E1 -16804.697,E2 -16804.697} C_VEL
LIN {X 0,Y 292.983,Z 582.58,A -85,B 0,C 180,E1 -16806.683,E2 -16806.683} C_VEL
LIN {X 0,Y 294.382,Z 573.265,A -85,B 0,C 180,E1 -16808.604,E2 -16808.604} C_VEL
LIN {X 0,Y 295.738,Z 563.65,A -85,B 0,C 180,E1 -16810.204,E2 -16810.204} C_VEL
LIN {X 0,Y 297.105,Z 552.261,A -85,B 0,C 180,E1 -16811.713,E2 -16811.713} C_VEL
LIN {X 0,Y 298.443,Z 540.157,A -85,B 0,C 180,E1 -16812.967,E2 -16812.967} C_VEL
LIN {X 0,Y 299.473,Z 528.162,A -85,B 0,C 180,E1 -16813.906,E2 -16813.906} C_VEL
LIN {X 0,Y 300.391,Z 514.428,A -85,B 0,C 180,E1 -16814.666,E2 -16814.666} C_VEL
LIN {X 0,Y 300.972,Z 501.3,A -85,B 0,C 180,E1 -16815.114,E2 -16815.114} C_VEL
LIN {X 0,Y 302.909,Z 433.848,A -85,B 0,C 180,E1 -16816.818,E2 -16816.818} C_VEL
LIN {X 0,Y 300.744,Z 423.334,A -85,B 0,C 180,E1 -16817.27,E2 -16817.27} C_VEL
LIN {X 0,Y 293.381,Z 403.161,A -85,B 0,C 180,E1 -16818.418,E2 -16818.418} C_VEL
LIN {X 0,Y 292.672,Z 400.961,A -85,B 0,C 180,E1 -16818.567,E2 -16818.567} C_VEL
LIN {X 0,Y 291.645,Z 395.158,A -85,B 0,C 180,E1 -16820.731,E2 -16820.731} C_VEL
LIN {X 0,Y 291.702,Z 395.149,A -85,B 0,C 180,E1 -16823.079,E2 -16823.079} C_VEL
LIN {X 0,Y 291.792,Z 395.137,A -85,B 0,C 180,E1 -16827.237,E2 -16827.237} C_VEL
LIN {X 0,Y 291.969,Z 395.116,A -85,B 0,C 180,E1 -16829.998,E2 -16829.998} C_VEL
LIN {X 0,Y 291.793,Z 395.135,A -85,B 0,C 180,E1 -16832.759,E2 -16832.759} C_VEL
LIN {X 0,Y 291.749,Z 395.14,A -85,B 0,C 180,E1 -16836.916,E2 -16836.916} C_VEL
LIN {X 0,Y 291.631,Z 395.158,A -85,B 0,C 180,E1 -16839.71,E2 -16839.71} C_VEL
LIN {X 0,Y 291.523,Z 395.171,A -85,B 0,C 180,E1 -16843.948,E2 -16843.948} C_VEL
LIN {X 0,Y 291.488,Z 395.174,A -85,B 0,C 180,E1 -16846.816,E2 -16846.816} C_VEL
LIN {X 0,Y 291.45,Z 395.178,A -85,B 0,C 180,E1 -16849.873,E2 -16849.873} C_VEL
LIN {X 0,Y 291.397,Z 395.186,A -85,B 0,C 180,E1 -16854.203,E2 -16854.203} C_VEL
LIN {X 0,Y 291.421,Z 395.178,A -85,B 0,C 180,E1 -16857.269,E2 -16857.269} C_VEL
LIN {X 0,Y 291.337,Z 395.192,A -85,B 0,C 180,E1 -16860.434,E2 -16860.434} C_VEL
LIN {X 0,Y 291.342,Z 395.196,A -85,B 0,C 180,E1 -16863.696,E2 -16863.696} C_VEL
LIN {X 0,Y 291.4,Z 395.187,A -85,B 0,C 180,E1 -16867.26,E2 -16867.26} C_VEL
LIN {X 0,Y 291.373,Z 395.188,A -85,B 0,C 180,E1 -16870.633,E2 -16870.633} C_VEL
LIN {X 0,Y 291.408,Z 395.258,A -85,B 0,C 180,E1 -16871.978,E2 -16871.978} C_VEL
LIN {X 0,Y 292.076,Z 398.587,A -85,B 0,C 180,E1 -16872.881,E2 -16872.881} C_VEL
LIN {X 0,Y 298.212,Z 418.54,A -85,B 0,C 180,E1 -16873.912,E2 -16873.912} C_VEL
LIN {X 0,Y 300.488,Z 432.715,A -85,B 0,C 180,E1 -16874.492,E2 -16874.492} C_VEL
LIN {X 0,Y 298.583,Z 490.102,A -85,B 0,C 180,E1 -16876.198,E2 -16876.198} C_VEL
LIN {X 0,Y 297.616,Z 495.909,A -85,B 0,C 180,E1 -16876.33,E2 -16876.33} C_VEL
LIN {X 0,Y 291.656,Z 512.676,A -85,B 0,C 180,E1 -16876.683,E2 -16876.683} C_VEL
LIN {X 0,Y 290.494,Z 518.322,A -85,B 0,C 180,E1 -16876.93,E2 -16876.93} C_VEL
LIN {X 0,Y 290.413,Z 520.213,A -85,B 0,C 180,E1 -16877.039,E2 -16877.039} C_VEL
LIN {X 0,Y 289.588,Z 532.649,A -85,B 0,C 180,E1 -16877.899,E2 -16877.899} C_VEL
LIN {X 0,Y 288.453,Z 545.905,A -85,B 0,C 180,E1 -16879.134,E2 -16879.134} C_VEL
LIN {X 0,Y 287.354,Z 557.295,A -85,B 0,C 180,E1 -16880.513,E2 -16880.513} C_VEL
LIN {X 0,Y 286.163,Z 567.939,A -85,B 0,C 180,E1 -16882.121,E2 -16882.121} C_VEL
LIN {X 0,Y 285.057,Z 577.761,A -85,B 0,C 180,E1 -16883.963,E2 -16883.963} C_VEL
LIN {X 0,Y 284.248,Z 585.599,A -85,B 0,C 180,E1 -16885.771,E2 -16885.771} C_VEL
LIN {X 0,Y 283.442,Z 593.396,A -85,B 0,C 180,E1 -16887.995,E2 -16887.995} C_VEL
LIN {X 0,Y 282.862,Z 599.495,A -85,B 0,C 180,E1 -16890.203,E2 -16890.203} C_VEL
LIN {X 0,Y 282.517,Z 604.545,A -85,B 0,C 180,E1 -16892.599,E2 -16892.599} C_VEL
LIN {X 0,Y 282.151,Z 608.143,A -85,B 0,C 180,E1 -16894.947,E2 -16894.947} C_VEL
LIN {X 0,Y 282.015,Z 610.448,A -85,B 0,C 180,E1 -16897.224,E2 -16897.224} C_VEL
LIN {X 0,Y 282.063,Z 611.675,A -85,B 0,C 180,E1 -16899.584,E2 -16899.584} C_VEL
LIN {X 0,Y 282.268,Z 611.82,A -85,B 0,C 180,E1 -16901.114,E2 -16901.114} C_VEL
LIN {X 0,Y 282.474,Z 611.516,A -85,B 0,C 180,E1 -16902.629,E2 -16902.629} C_VEL
LIN {X 0,Y 282.755,Z 610.747,A -85,B 0,C 180,E1 -16904.133,E2 -16904.133} C_VEL
LIN {X 0,Y 283.196,Z 609.484,A -85,B 0,C 180,E1 -16905.631,E2 -16905.631} C_VEL
LIN {X 0,Y 284.037,Z 606.745,A -85,B 0,C 180,E1 -16907.859,E2 -16907.859} C_VEL
LIN {X 0,Y 285.283,Z 602.65,A -85,B 0,C 180,E1 -16910.186,E2 -16910.186} C_VEL
LIN {X 0,Y 286.961,Z 596.829,A -85,B 0,C 180,E1 -16912.612,E2 -16912.612} C_VEL
LIN {X 0,Y 288.815,Z 590.114,A -85,B 0,C 180,E1 -16914.761,E2 -16914.761} C_VEL
LIN {X 0,Y 291.068,Z 581.778,A -85,B 0,C 180,E1 -16916.886,E2 -16916.886} C_VEL
LIN {X 0,Y 293.174,Z 573.218,A -85,B 0,C 180,E1 -16918.626,E2 -16918.626} C_VEL
LIN {X 0,Y 295.653,Z 562.502,A -85,B 0,C 180,E1 -16920.369,E2 -16920.369} C_VEL
LIN {X 0,Y 297.694,Z 552.336,A -85,B 0,C 180,E1 -16921.691,E2 -16921.691} C_VEL
LIN {X 0,Y 299.961,Z 539.243,A -85,B 0,C 180,E1 -16923.022,E2 -16923.022} C_VEL
LIN {X 0,Y 301.705,Z 526.451,A -85,B 0,C 180,E1 -16924.007,E2 -16924.007} C_VEL
LIN {X 0,Y 303.19,Z 512.872,A -85,B 0,C 180,E1 -16924.746,E2 -16924.746} C_VEL
LIN {X 0,Y 305.095,Z 484.748,A -85,B 0,C 180,E1 -16925.701,E2 -16925.701} C_VEL
LIN {X 0,Y 308.028,Z 440.126,A -85,B 0,C 180,E1 -16927.172,E2 -16927.172} C_VEL
LIN {X 0,Y 304.892,Z 432.833,A -85,B 0,C 180,E1 -16928.067,E2 -16928.067} C_VEL
LIN {X 0,Y 299.696,Z 422.084,A -85,B 0,C 180,E1 -16929.58,E2 -16929.58} C_VEL
LIN {X 0,Y 295.516,Z 414.897,A -85,B 0,C 180,E1 -16930.851,E2 -16930.851} C_VEL
LIN {X 0,Y 292.09,Z 409.664,A -85,B 0,C 180,E1 -16931.935,E2 -16931.935} C_VEL
LIN {X 0,Y 286.376,Z 401.269,A -85,B 0,C 180,E1 -16933.935,E2 -16933.935} C_VEL
LIN {X 0,Y 285.727,Z 399.237,A -85,B 0,C 180,E1 -16934.858,E2 -16934.858} C_VEL
LIN {X 0,Y 284.457,Z 396.053,A -85,B 0,C 180,E1 -16936.534,E2 -16936.534} C_VEL
LIN {X 0,Y 284.417,Z 396.058,A -85,B 0,C 180,E1 -16940.239,E2 -16940.239} C_VEL
LIN {X 0,Y 284.391,Z 396.061,A -85,B 0,C 180,E1 -16943.891,E2 -16943.891} C_VEL
LIN {X 0,Y 284.323,Z 396.067,A -85,B 0,C 180,E1 -16948.012,E2 -16948.012} C_VEL
LIN {X 0,Y 284.289,Z 396.072,A -85,B 0,C 180,E1 -16951.275,E2 -16951.275} C_VEL
LIN {X 0,Y 284.353,Z 396.063,A -85,B 0,C 180,E1 -16955.355,E2 -16955.355} C_VEL
LIN {X 0,Y 284.315,Z 396.07,A -85,B 0,C 180,E1 -16958.169,E2 -16958.169} C_VEL
LIN {X 0,Y 284.289,Z 396.072,A -85,B 0,C 180,E1 -16962.132,E2 -16962.132} C_VEL
LIN {X 0,Y 284.261,Z 396.074,A -85,B 0,C 180,E1 -16966.193,E2 -16966.193} C_VEL
LIN {X 0,Y 284.3,Z 396.072,A -85,B 0,C 180,E1 -16970.026,E2 -16970.026} C_VEL
LIN {X 0,Y 284.318,Z 396.166,A -85,B 0,C 180,E1 -16971.524,E2 -16971.524} C_VEL
LIN {X 0,Y 284.854,Z 398.048,A -85,B 0,C 180,E1 -16972.14,E2 -16972.14} C_VEL
LIN {X 0,Y 286.84,Z 401.116,A -85,B 0,C 180,E1 -16973.392,E2 -16973.392} C_VEL
LIN {X 0,Y 289.427,Z 405.921,A -85,B 0,C 180,E1 -16974.96,E2 -16974.96} C_VEL
LIN {X 0,Y 294.295,Z 413.263,A -85,B 0,C 180,E1 -16976.57,E2 -16976.57} C_VEL
LIN {X 0,Y 298.089,Z 421.901,A -85,B 0,C 180,E1 -16977.862,E2 -16977.862} C_VEL
LIN {X 0,Y 302.321,Z 432.479,A -85,B 0,C 180,E1 -16979.243,E2 -16979.243} C_VEL
LIN {X 0,Y 303.623,Z 437.103,A -85,B 0,C 180,E1 -16979.703,E2 -16979.703} C_VEL
LIN {X 0,Y 305.988,Z 456.231,A -85,B 0,C 180,E1 -16981.005,E2 -16981.005} C_VEL
LIN {X 0,Y 306.308,Z 463.52,A -85,B 0,C 180,E1 -16981.392,E2 -16981.392} C_VEL
LIN {X 0,Y 302.211,Z 524.939,A -85,B 0,C 180,E1 -16983.455,E2 -16983.455} C_VEL
LIN {X 0,Y 300.547,Z 539.171,A -85,B 0,C 180,E1 -16984.183,E2 -16984.183} C_VEL
LIN {X 0,Y 298.587,Z 551.866,A -85,B 0,C 180,E1 -16985.121,E2 -16985.121} C_VEL
LIN {X 0,Y 296.256,Z 564.866,A -85,B 0,C 180,E1 -16986.404,E2 -16986.404} C_VEL
LIN {X 0,Y 293.855,Z 576.309,A -85,B 0,C 180,E1 -16987.874,E2 -16987.874} C_VEL
LIN {X 0,Y 291.501,Z 586.618,A -85,B 0,C 180,E1 -16989.54,E2 -16989.54} C_VEL
LIN {X 0,Y 289.084,Z 596.516,A -85,B 0,C 180,E1 -16991.578,E2 -16991.578} C_VEL
LIN {X 0,Y 287.217,Z 604.562,A -85,B 0,C 180,E1 -16993.658,E2 -16993.658} C_VEL
LIN {X 0,Y 285.464,Z 611.04,A -85,B 0,C 180,E1 -16995.75,E2 -16995.75} C_VEL
LIN {X 0,Y 284.181,Z 616.198,A -85,B 0,C 180,E1 -16997.867,E2 -16997.867} C_VEL
LIN {X 0,Y 283.297,Z 620.192,A -85,B 0,C 180,E1 -17000.002,E2 -17000.002} C_VEL
LIN {X 0,Y 282.878,Z 622.274,A -85,B 0,C 180,E1 -17001.429,E2 -17001.429} C_VEL
LIN {X 0,Y 282.599,Z 623.928,A -85,B 0,C 180,E1 -17002.859,E2 -17002.859} C_VEL
LIN {X 0,Y 282.425,Z 625.233,A -85,B 0,C 180,E1 -17004.49,E2 -17004.49} C_VEL
LIN {X 0,Y 282.364,Z 626.382,A -85,B 0,C 180,E1 -17007.149,E2 -17007.149} C_VEL
LIN {X 0,Y 282.339,Z 627.316,A -85,B 0,C 180,E1 -17008.576,E2 -17008.576} C_VEL
LIN {X 0,Y 282.355,Z 627.847,A -85,B 0,C 180,E1 -17010.002,E2 -17010.002} C_VEL
LIN {X 0,Y 282.33,Z 627.93,A -85,B 0,C 180,E1 -17011.428,E2 -17011.428} C_VEL
LIN {X 0,Y 282.336,Z 627.609,A -85,B 0,C 180,E1 -17012.855,E2 -17012.855} C_VEL
LIN {X 0,Y 282.386,Z 625.783,A -85,B 0,C 180,E1 -17015.715,E2 -17015.715} C_VEL
LIN {X 0,Y 282.558,Z 624.215,A -85,B 0,C 180,E1 -17017.146,E2 -17017.146} C_VEL
LIN {X 0,Y 283.038,Z 621.081,A -85,B 0,C 180,E1 -17019.29,E2 -17019.29} C_VEL
LIN {X 0,Y 283.791,Z 616.891,A -85,B 0,C 180,E1 -17021.429,E2 -17021.429} C_VEL
LIN {X 0,Y 285.078,Z 610.513,A -85,B 0,C 180,E1 -17023.91,E2 -17023.91} C_VEL
LIN {X 0,Y 286.703,Z 603.591,A -85,B 0,C 180,E1 -17026.01,E2 -17026.01} C_VEL
LIN {X 0,Y 288.074,Z 596.633,A -85,B 0,C 180,E1 -17027.739,E2 -17027.739} C_VEL
LIN {X 0,Y 289.817,Z 588.117,A -85,B 0,C 180,E1 -17029.479,E2 -17029.479} C_VEL
LIN {X 0,Y 291.942,Z 577.732,A -85,B 0,C 180,E1 -17031.169,E2 -17031.169} C_VEL
LIN {X 0,Y 294.073,Z 566.109,A -85,B 0,C 180,E1 -17032.668,E2 -17032.668} C_VEL
LIN {X 0,Y 295.811,Z 554.689,A -85,B 0,C 180,E1 -17033.823,E2 -17033.823} C_VEL
LIN {X 0,Y 297.511,Z 541.722,A -85,B 0,C 180,E1 -17034.792,E2 -17034.792} C_VEL
LIN {X 0,Y 298.872,Z 528.862,A -85,B 0,C 180,E1 -17035.462,E2 -17035.462} C_VEL
LIN {X 0,Y 299.613,Z 515.474,A -85,B 0,C 180,E1 -17035.907,E2 -17035.907} C_VEL
LIN {X 0,Y 301.591,Z 460.997,A -85,B 0,C 180,E1 -17037.345,E2 -17037.345} C_VEL
LIN {X 0,Y 298.879,Z 442.5,A -85,B 0,C 180,E1 -17038.257,E2 -17038.257} C_VEL
LIN {X 0,Y 296.7,Z 431.949,A -85,B 0,C 180,E1 -17038.874,E2 -17038.874} C_VEL
LIN {X 0,Y 290.831,Z 418.71,A -85,B 0,C 180,E1 -17040.116,E2 -17040.116} C_VEL
LIN {X 0,Y 288.85,Z 414.566,A -85,B 0,C 180,E1 -17040.57,E2 -17040.57} C_VEL
LIN {X 0,Y 286.736,Z 405.082,A -85,B 0,C 180,E1 -17044.317,E2 -17044.317} C_VEL
LIN {X 0,Y 285.005,Z 398.481,A -85,B 0,C 180,E1 -17047.17,E2 -17047.17} C_VEL
LIN {X 0,Y 284.349,Z 396.069,A -85,B 0,C 180,E1 -17048.278,E2 -17048.278} C_VEL
LIN {X 0,Y 284.275,Z 396.077,A -85,B 0,C 180,E1 -17052.125,E2 -17052.125} C_VEL
LIN {X 0,Y 284.261,Z 396.079,A -85,B 0,C 180,E1 -17056.19,E2 -17056.19} C_VEL
LIN {X 0,Y 284.312,Z 396.063,A -85,B 0,C 180,E1 -17060.025,E2 -17060.025} C_VEL
LIN {X 0,Y 284.338,Z 396.063,A -85,B 0,C 180,E1 -17063.615,E2 -17063.615} C_VEL
LIN {X 0,Y 284.314,Z 396.067,A -85,B 0,C 180,E1 -17067.19,E2 -17067.19} C_VEL
LIN {X 0,Y 284.362,Z 396.056,A -85,B 0,C 180,E1 -17070.376,E2 -17070.376} C_VEL
LIN {X 0,Y 284.381,Z 396.051,A -85,B 0,C 180,E1 -17073.587,E2 -17073.587} C_VEL
LIN {X 0,Y 284.373,Z 396.053,A -85,B 0,C 180,E1 -17076.708,E2 -17076.708} C_VEL
LIN {X 0,Y 284.41,Z 396.046,A -85,B 0,C 180,E1 -17081.262,E2 -17081.262} C_VEL
LIN {X 0,Y 284.499,Z 396.04,A -85,B 0,C 180,E1 -17084.46,E2 -17084.46} C_VEL
LIN {X 0,Y 284.495,Z 396.04,A -85,B 0,C 180,E1 -17088.602,E2 -17088.602} C_VEL
LIN {X 0,Y 284.667,Z 396.026,A -85,B 0,C 180,E1 -17091.481,E2 -17091.481} C_VEL
LIN {X 0,Y 284.608,Z 396.028,A -85,B 0,C 180,E1 -17094.332,E2 -17094.332} C_VEL
LIN {X 0,Y 284.861,Z 396.003,A -85,B 0,C 180,E1 -17098.586,E2 -17098.586} C_VEL
LIN {X 0,Y 284.861,Z 395.998,A -85,B 0,C 180,E1 -17101.414,E2 -17101.414} C_VEL
LIN {X 0,Y 284.706,Z 396.017,A -85,B 0,C 180,E1 -17107.09,E2 -17107.09} C_VEL
LIN {X 0,Y 284.574,Z 396.036,A -85,B 0,C 180,E1 -17109.955,E2 -17109.955} C_VEL
LIN {X 0,Y 284.489,Z 396.046,A -85,B 0,C 180,E1 -17114.303,E2 -17114.303} C_VEL
LIN {X 0,Y 284.441,Z 396.075,A -85,B 0,C 180,E1 -17117.897,E2 -17117.897} C_VEL
LIN {X 0,Y 286.172,Z 403.089,A -85,B 0,C 180,E1 -17121.129,E2 -17121.129} C_VEL
LIN {X 0,Y 294.407,Z 418.714,A -85,B 0,C 180,E1 -17122.854,E2 -17122.854} C_VEL
LIN {X 0,Y 300.663,Z 432.781,A -85,B 0,C 180,E1 -17124.131,E2 -17124.131} C_VEL
LIN {X 0,Y 302.336,Z 437.272,A -85,B 0,C 180,E1 -17124.477,E2 -17124.477} C_VEL
LIN {X 0,Y 299.569,Z 509.842,A -85,B 0,C 180,E1 -17126.43,E2 -17126.43} C_VEL
LIN {X 0,Y 298.55,Z 522.848,A -85,B 0,C 180,E1 -17127.027,E2 -17127.027} C_VEL
LIN {X 0,Y 297.269,Z 535.123,A -85,B 0,C 180,E1 -17127.855,E2 -17127.855} C_VEL
LIN {X 0,Y 295.566,Z 547.691,A -85,B 0,C 180,E1 -17129.014,E2 -17129.014} C_VEL
LIN {X 0,Y 293.736,Z 558.816,A -85,B 0,C 180,E1 -17130.344,E2 -17130.344} C_VEL
LIN {X 0,Y 291.917,Z 568.576,A -85,B 0,C 180,E1 -17131.803,E2 -17131.803} C_VEL
LIN {X 0,Y 289.889,Z 578.375,A -85,B 0,C 180,E1 -17133.632,E2 -17133.632} C_VEL
LIN {X 0,Y 287.988,Z 586.729,A -85,B 0,C 180,E1 -17135.577,E2 -17135.577} C_VEL
LIN {X 0,Y 286.172,Z 594.558,A -85,B 0,C 180,E1 -17137.877,E2 -17137.877} C_VEL
LIN {X 0,Y 284.87,Z 600.412,A -85,B 0,C 180,E1 -17140.109,E2 -17140.109} C_VEL
LIN {X 0,Y 283.988,Z 604.447,A -85,B 0,C 180,E1 -17142.059,E2 -17142.059} C_VEL
LIN {X 0,Y 283.269,Z 607.555,A -85,B 0,C 180,E1 -17144.003,E2 -17144.003} C_VEL
LIN {X 0,Y 282.643,Z 610.005,A -85,B 0,C 180,E1 -17146.145,E2 -17146.145} C_VEL
LIN {X 0,Y 282.276,Z 611.525,A -85,B 0,C 180,E1 -17148.325,E2 -17148.325} C_VEL
LIN {X 0,Y 282.055,Z 612.112,A -85,B 0,C 180,E1 -17150.573,E2 -17150.573} C_VEL
LIN {X 0,Y 282.013,Z 611.519,A -85,B 0,C 180,E1 -17153.264,E2 -17153.264} C_VEL
LIN {X 0,Y 282.159,Z 610.109,A -85,B 0,C 180,E1 -17155.282,E2 -17155.282} C_VEL
LIN {X 0,Y 282.562,Z 607.254,A -85,B 0,C 180,E1 -17157.743,E2 -17157.743} C_VEL
LIN {X 0,Y 283.13,Z 602.789,A -85,B 0,C 180,E1 -17160.319,E2 -17160.319} C_VEL
LIN {X 0,Y 283.799,Z 597.718,A -85,B 0,C 180,E1 -17162.503,E2 -17162.503} C_VEL
LIN {X 0,Y 284.822,Z 590.874,A -85,B 0,C 180,E1 -17164.807,E2 -17164.807} C_VEL
LIN {X 0,Y 285.943,Z 583.216,A -85,B 0,C 180,E1 -17166.841,E2 -17166.841} C_VEL
LIN {X 0,Y 287.421,Z 573.732,A -85,B 0,C 180,E1 -17168.857,E2 -17168.857} C_VEL
LIN {X 0,Y 288.877,Z 563.832,A -85,B 0,C 180,E1 -17170.547,E2 -17170.547} C_VEL
LIN {X 0,Y 290.201,Z 553.089,A -85,B 0,C 180,E1 -17172.013,E2 -17172.013} C_VEL
LIN {X 0,Y 291.614,Z 541.03,A -85,B 0,C 180,E1 -17173.303,E2 -17173.303} C_VEL
LIN {X 0,Y 292.644,Z 529.711,A -85,B 0,C 180,E1 -17174.236,E2 -17174.236} C_VEL
LIN {X 0,Y 293.556,Z 516.496,A -85,B 0,C 180,E1 -17175.018,E2 -17175.018} C_VEL
LIN {X 0,Y 294.182,Z 503.334,A -85,B 0,C 180,E1 -17175.515,E2 -17175.515} C_VEL
LIN {X 0,Y 296.214,Z 434.6,A -85,B 0,C 180,E1 -17177.296,E2 -17177.296} C_VEL
LIN {X 0,Y 294.314,Z 425.394,A -85,B 0,C 180,E1 -17177.705,E2 -17177.705} C_VEL
LIN {X 0,Y 286.411,Z 403.781,A -85,B 0,C 180,E1 -17178.972,E2 -17178.972} C_VEL
LIN {X 0,Y 285.533,Z 401.18,A -85,B 0,C 180,E1 -17179.148,E2 -17179.148} C_VEL
LIN {X 0,Y 284.633,Z 396.03,A -85,B 0,C 180,E1 -17181.09,E2 -17181.09} C_VEL
LIN {X 0,Y 284.585,Z 396.037,A -85,B 0,C 180,E1 -17184.329,E2 -17184.329} C_VEL
LIN {X 0,Y 284.858,Z 396.003,A -85,B 0,C 180,E1 -17188.584,E2 -17188.584} C_VEL
LIN {X 0,Y 284.859,Z 396.001,A -85,B 0,C 180,E1 -17191.412,E2 -17191.412} C_VEL
LIN {X 0,Y 284.701,Z 396.017,A -85,B 0,C 180,E1 -17197.088,E2 -17197.088} C_VEL
LIN {X 0,Y 284.568,Z 396.04,A -85,B 0,C 180,E1 -17199.953,E2 -17199.953} C_VEL
LIN {X 0,Y 284.482,Z 396.05,A -85,B 0,C 180,E1 -17204.301,E2 -17204.301} C_VEL
LIN {X 0,Y 284.426,Z 396.054,A -85,B 0,C 180,E1 -17207.246,E2 -17207.246} C_VEL
LIN {X 0,Y 284.377,Z 396.06,A -85,B 0,C 180,E1 -17210.24,E2 -17210.24} C_VEL
LIN {X 0,Y 284.366,Z 396.065,A -85,B 0,C 180,E1 -17213.872,E2 -17213.872} C_VEL
LIN {X 0,Y 284.395,Z 396.053,A -85,B 0,C 180,E1 -17217.172,E2 -17217.172} C_VEL
LIN {X 0,Y 284.296,Z 396.07,A -85,B 0,C 180,E1 -17221.272,E2 -17221.272} C_VEL
LIN {X 0,Y 284.358,Z 396.064,A -85,B 0,C 180,E1 -17225.352,E2 -17225.352} C_VEL
LIN {X 0,Y 284.33,Z 396.067,A -85,B 0,C 180,E1 -17228.163,E2 -17228.163} C_VEL
LIN {X 0,Y 284.377,Z 396.193,A -85,B 0,C 180,E1 -17231.735,E2 -17231.735} C_VEL
LIN {X 0,Y 284.868,Z 398.766,A -85,B 0,C 180,E1 -17232.43,E2 -17232.43} C_VEL
LIN {X 0,Y 291.555,Z 420.384,A -85,B 0,C 180,E1 -17233.584,E2 -17233.584} C_VEL
LIN {X 0,Y 293.66,Z 433.913,A -85,B 0,C 180,E1 -17234.149,E2 -17234.149} C_VEL
LIN {X 0,Y 290.968,Z 509.306,A -85,B 0,C 180,E1 -17236.496,E2 -17236.496} C_VEL
LIN {X 0,Y 290.413,Z 520.213,A -85,B 0,C 180,E1 -17237.039,E2 -17237.039} C_VEL
LIN {X 0,Y 289.607,Z 523.978,A -85,B 0,C 180,E1 -17237.239,E2 -17237.239} C_VEL
LIN {X 0,Y 286.381,Z 529.76,A -85,B 0,C 180,E1 -17237.519,E2 -17237.519} C_VEL
LIN {X 0,Y 283.056,Z 535.42,A -85,B 0,C 180,E1 -17237.866,E2 -17237.866} C_VEL
LIN {X 0,Y 282.125,Z 539,A -85,B 0,C 180,E1 -17238.171,E2 -17238.171} C_VEL
LIN {X 0,Y 280.979,Z 550.788,A -85,B 0,C 180,E1 -17239.433,E2 -17239.433} C_VEL
LIN {X 0,Y 279.883,Z 561.485,A -85,B 0,C 180,E1 -17240.883,E2 -17240.883} C_VEL
LIN {X 0,Y 278.685,Z 572.52,A -85,B 0,C 180,E1 -17242.753,E2 -17242.753} C_VEL
LIN {X 0,Y 277.705,Z 580.477,A -85,B 0,C 180,E1 -17244.403,E2 -17244.403} C_VEL
LIN {X 0,Y 276.844,Z 588.973,A -85,B 0,C 180,E1 -17246.57,E2 -17246.57} C_VEL
LIN {X 0,Y 276.071,Z 596.44,A -85,B 0,C 180,E1 -17248.968,E2 -17248.968} C_VEL
LIN {X 0,Y 275.651,Z 601.48,A -85,B 0,C 180,E1 -17251.025,E2 -17251.025} C_VEL
LIN {X 0,Y 275.293,Z 605.814,A -85,B 0,C 180,E1 -17253.314,E2 -17253.314} C_VEL
LIN {X 0,Y 274.954,Z 609.208,A -85,B 0,C 180,E1 -17255.86,E2 -17255.86} C_VEL
LIN {X 0,Y 274.916,Z 610.667,A -85,B 0,C 180,E1 -17257.451,E2 -17257.451} C_VEL
LIN {X 0,Y 274.913,Z 611.578,A -85,B 0,C 180,E1 -17259.028,E2 -17259.028} C_VEL
LIN {X 0,Y 275.151,Z 612.048,A -85,B 0,C 180,E1 -17260.913,E2 -17260.913} C_VEL
LIN {X 0,Y 275.306,Z 611.966,A -85,B 0,C 180,E1 -17262.161,E2 -17262.161} C_VEL
LIN {X 0,Y 275.581,Z 611.419,A -85,B 0,C 180,E1 -17263.708,E2 -17263.708} C_VEL
LIN {X 0,Y 276.01,Z 610.352,A -85,B 0,C 180,E1 -17265.363,E2 -17265.363} C_VEL
LIN {X 0,Y 276.504,Z 608.994,A -85,B 0,C 180,E1 -17266.776,E2 -17266.776} C_VEL
LIN {X 0,Y 277.529,Z 605.909,A -85,B 0,C 180,E1 -17269.051,E2 -17269.051} C_VEL
LIN {X 0,Y 278.919,Z 601.661,A -85,B 0,C 180,E1 -17271.304,E2 -17271.304} C_VEL
LIN {X 0,Y 280.943,Z 595.18,A -85,B 0,C 180,E1 -17273.897,E2 -17273.897} C_VEL
LIN {X 0,Y 283.084,Z 588.002,A -85,B 0,C 180,E1 -17276.085,E2 -17276.085} C_VEL
LIN {X 0,Y 285.577,Z 579.067,A -85,B 0,C 180,E1 -17278.237,E2 -17278.237} C_VEL
LIN {X 0,Y 288.137,Z 569.095,A -85,B 0,C 180,E1 -17280.121,E2 -17280.121} C_VEL
LIN {X 0,Y 290.589,Z 558.501,A -85,B 0,C 180,E1 -17281.732,E2 -17281.732} C_VEL
LIN {X 0,Y 292.9,Z 547.12,A -85,B 0,C 180,E1 -17283.095,E2 -17283.095} C_VEL
LIN {X 0,Y 294.984,Z 534.686,A -85,B 0,C 180,E1 -17284.253,E2 -17284.253} C_VEL
LIN {X 0,Y 296.688,Z 521.698,A -85,B 0,C 180,E1 -17285.152,E2 -17285.152} C_VEL
LIN {X 0,Y 298.03,Z 508.246,A -85,B 0,C 180,E1 -17285.79,E2 -17285.79} C_VEL
LIN {X 0,Y 302.708,Z 442.501,A -85,B 0,C 180,E1 -17288.007,E2 -17288.007} C_VEL
LIN {X 0,Y 296.428,Z 428.468,A -85,B 0,C 180,E1 -17289.933,E2 -17289.933} C_VEL
LIN {X 0,Y 291.857,Z 420.388,A -85,B 0,C 180,E1 -17291.371,E2 -17291.371} C_VEL
LIN {X 0,Y 288.105,Z 414.434,A -85,B 0,C 180,E1 -17292.653,E2 -17292.653} C_VEL
LIN {X 0,Y 282.862,Z 406.706,A -85,B 0,C 180,E1 -17294.587,E2 -17294.587} C_VEL
LIN {X 0,Y 279.184,Z 401.423,A -85,B 0,C 180,E1 -17296.179,E2 -17296.179} C_VEL
LIN {X 0,Y 277.374,Z 396.936,A -85,B 0,C 180,E1 -17298.848,E2 -17298.848} C_VEL
LIN {X 0,Y 277.315,Z 396.941,A -85,B 0,C 180,E1 -17302.343,E2 -17302.343} C_VEL
LIN {X 0,Y 277.316,Z 396.943,A -85,B 0,C 180,E1 -17305.52,E2 -17305.52} C_VEL
LIN {X 0,Y 277.281,Z 396.947,A -85,B 0,C 180,E1 -17308.788,E2 -17308.788} C_VEL
LIN {X 0,Y 277.247,Z 396.948,A -85,B 0,C 180,E1 -17313.229,E2 -17313.229} C_VEL
LIN {X 0,Y 277.316,Z 396.941,A -85,B 0,C 180,E1 -17315.813,E2 -17315.813} C_VEL
LIN {X 0,Y 277.246,Z 396.949,A -85,B 0,C 180,E1 -17319.326,E2 -17319.326} C_VEL
LIN {X 0,Y 277.226,Z 396.953,A -85,B 0,C 180,E1 -17323.195,E2 -17323.195} C_VEL
LIN {X 0,Y 277.211,Z 396.953,A -85,B 0,C 180,E1 -17327.326,E2 -17327.326} C_VEL
LIN {X 0,Y 277.225,Z 397.07,A -85,B 0,C 180,E1 -17329.148,E2 -17329.148} C_VEL
LIN {X 0,Y 278.281,Z 399.802,A -85,B 0,C 180,E1 -17330.307,E2 -17330.307} C_VEL
LIN {X 0,Y 279.631,Z 401.372,A -85,B 0,C 180,E1 -17331.181,E2 -17331.181} C_VEL
LIN {X 0,Y 281.196,Z 404.652,A -85,B 0,C 180,E1 -17332.441,E2 -17332.441} C_VEL
LIN {X 0,Y 282.545,Z 406.618,A -85,B 0,C 180,E1 -17333.088,E2 -17333.088} C_VEL
LIN {X 0,Y 286.138,Z 411.718,A -85,B 0,C 180,E1 -17334.444,E2 -17334.444} C_VEL
LIN {X 0,Y 290.365,Z 418.192,A -85,B 0,C 180,E1 -17335.923,E2 -17335.923} C_VEL
LIN {X 0,Y 294.116,Z 427.105,A -85,B 0,C 180,E1 -17337.291,E2 -17337.291} C_VEL
LIN {X 0,Y 297.885,Z 436.986,A -85,B 0,C 180,E1 -17338.595,E2 -17338.595} C_VEL
LIN {X 0,Y 298.697,Z 440.306,A -85,B 0,C 180,E1 -17338.925,E2 -17338.925} C_VEL
LIN {X 0,Y 300.734,Z 458.046,A -85,B 0,C 180,E1 -17340.177,E2 -17340.177} C_VEL
LIN {X 0,Y 301.005,Z 464.024,A -85,B 0,C 180,E1 -17340.506,E2 -17340.506} C_VEL
LIN {X 0,Y 296.593,Z 525.145,A -85,B 0,C 180,E1 -17342.625,E2 -17342.625} C_VEL
LIN {X 0,Y 294.877,Z 539.214,A -85,B 0,C 180,E1 -17343.363,E2 -17343.363} C_VEL
LIN {X 0,Y 292.924,Z 550.946,A -85,B 0,C 180,E1 -17344.225,E2 -17344.225} C_VEL
LIN {X 0,Y 290.508,Z 564.021,A -85,B 0,C 180,E1 -17345.528,E2 -17345.528} C_VEL
LIN {X 0,Y 287.922,Z 575.511,A -85,B 0,C 180,E1 -17347.013,E2 -17347.013} C_VEL
LIN {X 0,Y 285.405,Z 585.887,A -85,B 0,C 180,E1 -17348.704,E2 -17348.704} C_VEL
LIN {X 0,Y 283.226,Z 594.412,A -85,B 0,C 180,E1 -17350.431,E2 -17350.431} C_VEL
LIN {X 0,Y 281.03,Z 602.744,A -85,B 0,C 180,E1 -17352.539,E2 -17352.539} C_VEL
LIN {X 0,Y 279.181,Z 609.512,A -85,B 0,C 180,E1 -17354.675,E2 -17354.675} C_VEL
LIN {X 0,Y 277.6,Z 614.966,A -85,B 0,C 180,E1 -17356.831,E2 -17356.831} C_VEL
LIN {X 0,Y 276.551,Z 619.216,A -85,B 0,C 180,E1 -17359.014,E2 -17359.014} C_VEL
LIN {X 0,Y 275.835,Z 622.381,A -85,B 0,C 180,E1 -17361.208,E2 -17361.208} C_VEL
LIN {X 0,Y 275.527,Z 623.929,A -85,B 0,C 180,E1 -17362.675,E2 -17362.675} C_VEL
LIN {X 0,Y 275.322,Z 625.309,A -85,B 0,C 180,E1 -17364.583,E2 -17364.583} C_VEL
LIN {X 0,Y 275.271,Z 626.102,A -85,B 0,C 180,E1 -17367.075,E2 -17367.075} C_VEL
LIN {X 0,Y 275.264,Z 627.059,A -85,B 0,C 180,E1 -17368.539,E2 -17368.539} C_VEL
LIN {X 0,Y 275.277,Z 627.616,A -85,B 0,C 180,E1 -17370.002,E2 -17370.002} C_VEL
LIN {X 0,Y 275.255,Z 627.738,A -85,B 0,C 180,E1 -17371.465,E2 -17371.465} C_VEL
LIN {X 0,Y 275.245,Z 627.44,A -85,B 0,C 180,E1 -17372.929,E2 -17372.929} C_VEL
LIN {X 0,Y 275.301,Z 625.667,A -85,B 0,C 180,E1 -17375.863,E2 -17375.863} C_VEL
LIN {X 0,Y 275.498,Z 624.148,A -85,B 0,C 180,E1 -17377.33,E2 -17377.33} C_VEL
LIN {X 0,Y 275.998,Z 621.065,A -85,B 0,C 180,E1 -17379.529,E2 -17379.529} C_VEL
LIN {X 0,Y 276.807,Z 616.928,A -85,B 0,C 180,E1 -17381.721,E2 -17381.721} C_VEL
LIN {X 0,Y 278.2,Z 610.606,A -85,B 0,C 180,E1 -17384.261,E2 -17384.261} C_VEL
LIN {X 0,Y 279.89,Z 603.747,A -85,B 0,C 180,E1 -17386.41,E2 -17386.41} C_VEL
LIN {X 0,Y 281.663,Z 595.381,A -85,B 0,C 180,E1 -17388.528,E2 -17388.528} C_VEL
LIN {X 0,Y 283.555,Z 586.598,A -85,B 0,C 180,E1 -17390.305,E2 -17390.305} C_VEL
LIN {X 0,Y 285.861,Z 575.953,A -85,B 0,C 180,E1 -17392.022,E2 -17392.022} C_VEL
LIN {X 0,Y 287.816,Z 565.442,A -85,B 0,C 180,E1 -17393.38,E2 -17393.38} C_VEL
LIN {X 0,Y 289.685,Z 553.844,A -85,B 0,C 180,E1 -17394.55,E2 -17394.55} C_VEL
LIN {X 0,Y 291.451,Z 540.694,A -85,B 0,C 180,E1 -17395.535,E2 -17395.535} C_VEL
LIN {X 0,Y 292.873,Z 527.402,A -85,B 0,C 180,E1 -17396.213,E2 -17396.213} C_VEL
LIN {X 0,Y 293.718,Z 510.118,A -85,B 0,C 180,E1 -17396.754,E2 -17396.754} C_VEL
LIN {X 0,Y 295.516,Z 461.313,A -85,B 0,C 180,E1 -17398.079,E2 -17398.079} C_VEL
LIN {X 0,Y 292.963,Z 443.856,A -85,B 0,C 180,E1 -17398.984,E2 -17398.984} C_VEL
LIN {X 0,Y 291.213,Z 435.009,A -85,B 0,C 180,E1 -17399.517,E2 -17399.517} C_VEL
LIN {X 0,Y 285.612,Z 422.44,A -85,B 0,C 180,E1 -17400.748,E2 -17400.748} C_VEL
LIN {X 0,Y 281.631,Z 414.304,A -85,B 0,C 180,E1 -17401.677,E2 -17401.677} C_VEL
LIN {X 0,Y 279.626,Z 405.55,A -85,B 0,C 180,E1 -17405.317,E2 -17405.317} C_VEL
LIN {X 0,Y 277.48,Z 397.843,A -85,B 0,C 180,E1 -17408.882,E2 -17408.882} C_VEL
LIN {X 0,Y 277.295,Z 396.951,A -85,B 0,C 180,E1 -17409.32,E2 -17409.32} C_VEL
LIN {X 0,Y 277.215,Z 396.958,A -85,B 0,C 180,E1 -17413.199,E2 -17413.199} C_VEL
LIN {X 0,Y 277.221,Z 396.95,A -85,B 0,C 180,E1 -17417.326,E2 -17417.326} C_VEL
LIN {X 0,Y 277.271,Z 396.947,A -85,B 0,C 180,E1 -17421.793,E2 -17421.793} C_VEL
LIN {X 0,Y 277.291,Z 396.945,A -85,B 0,C 180,E1 -17424.342,E2 -17424.342} C_VEL
LIN {X 0,Y 277.25,Z 396.949,A -85,B 0,C 180,E1 -17427.837,E2 -17427.837} C_VEL
LIN {X 0,Y 277.293,Z 396.944,A -85,B 0,C 180,E1 -17431.213,E2 -17431.213} C_VEL
LIN {X 0,Y 277.318,Z 396.936,A -85,B 0,C 180,E1 -17434.48,E2 -17434.48} C_VEL
LIN {X 0,Y 277.292,Z 396.934,A -85,B 0,C 180,E1 -17437.655,E2 -17437.655} C_VEL
LIN {X 0,Y 277.352,Z 396.927,A -85,B 0,C 180,E1 -17440.767,E2 -17440.767} C_VEL
LIN {X 0,Y 277.442,Z 396.914,A -85,B 0,C 180,E1 -17445.326,E2 -17445.326} C_VEL
LIN {X 0,Y 277.514,Z 396.906,A -85,B 0,C 180,E1 -17449.789,E2 -17449.789} C_VEL
LIN {X 0,Y 277.66,Z 396.891,A -85,B 0,C 180,E1 -17452.729,E2 -17452.729} C_VEL
LIN {X 0,Y 277.827,Z 396.879,A -85,B 0,C 180,E1 -17458.551,E2 -17458.551} C_VEL
LIN {X 0,Y 277.827,Z 396.874,A -85,B 0,C 180,E1 -17461.45,E2 -17461.45} C_VEL
LIN {X 0,Y 277.661,Z 396.895,A -85,B 0,C 180,E1 -17467.271,E2 -17467.271} C_VEL
LIN {X 0,Y 277.514,Z 396.916,A -85,B 0,C 180,E1 -17470.211,E2 -17470.211} C_VEL
LIN {X 0,Y 277.442,Z 396.925,A -85,B 0,C 180,E1 -17474.674,E2 -17474.674} C_VEL
LIN {X 0,Y 277.408,Z 397.087,A -85,B 0,C 180,E1 -17476.939,E2 -17476.939} C_VEL
LIN {X 0,Y 278.974,Z 403.18,A -85,B 0,C 180,E1 -17479.979,E2 -17479.979} C_VEL
LIN {X 0,Y 280.996,Z 406.967,A -85,B 0,C 180,E1 -17480.449,E2 -17480.449} C_VEL
LIN {X 0,Y 287.454,Z 418.938,A -85,B 0,C 180,E1 -17481.877,E2 -17481.877} C_VEL
LIN {X 0,Y 294.058,Z 433.216,A -85,B 0,C 180,E1 -17483.284,E2 -17483.284} C_VEL
LIN {X 0,Y 296.448,Z 439.66,A -85,B 0,C 180,E1 -17483.814,E2 -17483.814} C_VEL
LIN {X 0,Y 293.432,Z 510.506,A -85,B 0,C 180,E1 -17485.746,E2 -17485.746} C_VEL
LIN {X 0,Y 292.335,Z 523.781,A -85,B 0,C 180,E1 -17486.377,E2 -17486.377} C_VEL
LIN {X 0,Y 290.992,Z 536.144,A -85,B 0,C 180,E1 -17487.245,E2 -17487.245} C_VEL
LIN {X 0,Y 289.237,Z 548.317,A -85,B 0,C 180,E1 -17488.404,E2 -17488.404} C_VEL
LIN {X 0,Y 287.351,Z 559.241,A -85,B 0,C 180,E1 -17489.741,E2 -17489.741} C_VEL
LIN {X 0,Y 285.274,Z 569.74,A -85,B 0,C 180,E1 -17491.362,E2 -17491.362} C_VEL
LIN {X 0,Y 283.032,Z 579.867,A -85,B 0,C 180,E1 -17493.348,E2 -17493.348} C_VEL
LIN {X 0,Y 280.972,Z 588.381,A -85,B 0,C 180,E1 -17495.444,E2 -17495.444} C_VEL
LIN {X 0,Y 279.104,Z 595.921,A -85,B 0,C 180,E1 -17497.83,E2 -17497.83} C_VEL
LIN {X 0,Y 277.915,Z 600.964,A -85,B 0,C 180,E1 -17499.853,E2 -17499.853} C_VEL
LIN {X 0,Y 276.696,Z 606.11,A -85,B 0,C 180,E1 -17502.556,E2 -17502.556} C_VEL
LIN {X 0,Y 275.716,Z 609.878,A -85,B 0,C 180,E1 -17505.539,E2 -17505.539} C_VEL
LIN {X 0,Y 275.169,Z 611.871,A -85,B 0,C 180,E1 -17508.388,E2 -17508.388} C_VEL
LIN {X 0,Y 274.995,Z 612.306,A -85,B 0,C 180,E1 -17510.287,E2 -17510.287} C_VEL
LIN {X 0,Y 274.886,Z 612.013,A -85,B 0,C 180,E1 -17512.428,E2 -17512.428} C_VEL
LIN {X 0,Y 275.028,Z 610.631,A -85,B 0,C 180,E1 -17514.858,E2 -17514.858} C_VEL
LIN {X 0,Y 275.425,Z 607.716,A -85,B 0,C 180,E1 -17517.596,E2 -17517.596} C_VEL
LIN {X 0,Y 275.979,Z 603.877,A -85,B 0,C 180,E1 -17519.979,E2 -17519.979} C_VEL
LIN {X 0,Y 276.509,Z 599.699,A -85,B 0,C 180,E1 -17521.951,E2 -17521.951} C_VEL
LIN {X 0,Y 277.369,Z 594.03,A -85,B 0,C 180,E1 -17524.08,E2 -17524.08} C_VEL
LIN {X 0,Y 278.453,Z 587.028,A -85,B 0,C 180,E1 -17526.18,E2 -17526.18} C_VEL
LIN {X 0,Y 279.844,Z 578.14,A -85,B 0,C 180,E1 -17528.314,E2 -17528.314} C_VEL
LIN {X 0,Y 281.244,Z 568.958,A -85,B 0,C 180,E1 -17530.092,E2 -17530.092} C_VEL
LIN {X 0,Y 282.698,Z 558.584,A -85,B 0,C 180,E1 -17531.706,E2 -17531.706} C_VEL
LIN {X 0,Y 284.093,Z 547.633,A -85,B 0,C 180,E1 -17533.062,E2 -17533.062} C_VEL
LIN {X 0,Y 285.26,Z 536.793,A -85,B 0,C 180,E1 -17534.124,E2 -17534.124} C_VEL
LIN {X 0,Y 286.338,Z 524.169,A -85,B 0,C 180,E1 -17535.064,E2 -17535.064} C_VEL
LIN {X 0,Y 287.221,Z 510.536,A -85,B 0,C 180,E1 -17535.744,E2 -17535.744} C_VEL
LIN {X 0,Y 288.091,Z 484.287,A -85,B 0,C 180,E1 -17536.497,E2 -17536.497} C_VEL
LIN {X 0,Y 289.637,Z 435.825,A -85,B 0,C 180,E1 -17537.775,E2 -17537.775} C_VEL
LIN {X 0,Y 288.063,Z 427.952,A -85,B 0,C 180,E1 -17538.128,E2 -17538.128} C_VEL
LIN {X 0,Y 280.292,Z 406.67,A -85,B 0,C 180,E1 -17539.411,E2 -17539.411} C_VEL
LIN {X 0,Y 278.394,Z 401.442,A -85,B 0,C 180,E1 -17539.746,E2 -17539.746} C_VEL
LIN {X 0,Y 277.571,Z 396.91,A -85,B 0,C 180,E1 -17541.535,E2 -17541.535} C_VEL
LIN {X 0,Y 277.554,Z 396.913,A -85,B 0,C 180,E1 -17544.185,E2 -17544.185} C_VEL
LIN {X 0,Y 277.824,Z 396.88,A -85,B 0,C 180,E1 -17548.549,E2 -17548.549} C_VEL
LIN {X 0,Y 277.825,Z 396.877,A -85,B 0,C 180,E1 -17551.448,E2 -17551.448} C_VEL
LIN {X 0,Y 277.656,Z 396.895,A -85,B 0,C 180,E1 -17557.269,E2 -17557.269} C_VEL
LIN {X 0,Y 277.508,Z 396.92,A -85,B 0,C 180,E1 -17560.209,E2 -17560.209} C_VEL
LIN {X 0,Y 277.435,Z 396.926,A -85,B 0,C 180,E1 -17564.672,E2 -17564.672} C_VEL
LIN {X 0,Y 277.344,Z 396.931,A -85,B 0,C 180,E1 -17569.232,E2 -17569.232} C_VEL
LIN {X 0,Y 277.316,Z 396.94,A -85,B 0,C 180,E1 -17574.168,E2 -17574.168} C_VEL
LIN {X 0,Y 277.324,Z 396.934,A -85,B 0,C 180,E1 -17577.503,E2 -17577.503} C_VEL
LIN {X 0,Y 277.269,Z 396.944,A -85,B 0,C 180,E1 -17580.479,E2 -17580.479} C_VEL
LIN {X 0,Y 277.251,Z 396.95,A -85,B 0,C 180,E1 -17583.893,E2 -17583.893} C_VEL
LIN {X 0,Y 277.285,Z 396.946,A -85,B 0,C 180,E1 -17587.464,E2 -17587.464} C_VEL
LIN {X 0,Y 277.322,Z 396.995,A -85,B 0,C 180,E1 -17591.455,E2 -17591.455} C_VEL
LIN {X 0,Y 277.726,Z 399.061,A -85,B 0,C 180,E1 -17591.988,E2 -17591.988} C_VEL
LIN {X 0,Y 284.949,Z 422.397,A -85,B 0,C 180,E1 -17593.248,E2 -17593.248} C_VEL
LIN {X 0,Y 286.846,Z 433.755,A -85,B 0,C 180,E1 -17593.748,E2 -17593.748} C_VEL
LIN {X 0,Y 284.1,Z 508.937,A -85,B 0,C 180,E1 -17596.159,E2 -17596.159} C_VEL
LIN {X 0,Y 283.485,Z 520.984,A -85,B 0,C 180,E1 -17596.775,E2 -17596.775} C_VEL
LIN {X 0,Y 282.552,Z 533.622,A -85,B 0,C 180,E1 -17597.69,E2 -17597.69} C_VEL
LIN {X 0,Y 282.125,Z 539,A -85,B 0,C 180,E1 -17598.171,E2 -17598.171} C_VEL
LIN {X 0,Y 281.11,Z 544.301,A -85,B 0,C 180,E1 -17598.679,E2 -17598.679} C_VEL
LIN {X 0,Y 277.563,Z 552.531,A -85,B 0,C 180,E1 -17599.536,E2 -17599.536} C_VEL
LIN {X 0,Y 273.81,Z 560.426,A -85,B 0,C 180,E1 -17600.526,E2 -17600.526} C_VEL
LIN {X 0,Y 272.489,Z 565.072,A -85,B 0,C 180,E1 -17601.235,E2 -17601.235} C_VEL
LIN {X 0,Y 271.248,Z 575.599,A -85,B 0,C 180,E1 -17603.189,E2 -17603.189} C_VEL
LIN {X 0,Y 270.322,Z 584.003,A -85,B 0,C 180,E1 -17605.112,E2 -17605.112} C_VEL
LIN {X 0,Y 269.477,Z 591.558,A -85,B 0,C 180,E1 -17607.237,E2 -17607.237} C_VEL
LIN {X 0,Y 268.806,Z 598.292,A -85,B 0,C 180,E1 -17609.627,E2 -17609.627} C_VEL
LIN {X 0,Y 268.393,Z 603.267,A -85,B 0,C 180,E1 -17611.879,E2 -17611.879} C_VEL
LIN {X 0,Y 268.029,Z 607.395,A -85,B 0,C 180,E1 -17614.364,E2 -17614.364} C_VEL
LIN {X 0,Y 267.844,Z 610.171,A -85,B 0,C 180,E1 -17616.822,E2 -17616.822} C_VEL
LIN {X 0,Y 267.791,Z 611.342,A -85,B 0,C 180,E1 -17618.443,E2 -17618.443} C_VEL
LIN {X 0,Y 268.043,Z 612.176,A -85,B 0,C 180,E1 -17620.711,E2 -17620.711} C_VEL
LIN {X 0,Y 268.399,Z 611.975,A -85,B 0,C 180,E1 -17623.26,E2 -17623.26} C_VEL
LIN {X 0,Y 268.901,Z 610.981,A -85,B 0,C 180,E1 -17625.237,E2 -17625.237} C_VEL
LIN {X 0,Y 269.906,Z 608.379,A -85,B 0,C 180,E1 -17627.977,E2 -17627.977} C_VEL
LIN {X 0,Y 271.051,Z 605.245,A -85,B 0,C 180,E1 -17630.146,E2 -17630.146} C_VEL
LIN {X 0,Y 272.757,Z 600.434,A -85,B 0,C 180,E1 -17632.598,E2 -17632.598} C_VEL
LIN {X 0,Y 275.045,Z 593.525,A -85,B 0,C 180,E1 -17635.2,E2 -17635.2} C_VEL
LIN {X 0,Y 277.493,Z 585.769,A -85,B 0,C 180,E1 -17637.46,E2 -17637.46} C_VEL
LIN {X 0,Y 280.265,Z 576.241,A -85,B 0,C 180,E1 -17639.641,E2 -17639.641} C_VEL
LIN {X 0,Y 282.932,Z 566.377,A -85,B 0,C 180,E1 -17641.423,E2 -17641.423} C_VEL
LIN {X 0,Y 285.534,Z 555.367,A -85,B 0,C 180,E1 -17642.998,E2 -17642.998} C_VEL
LIN {X 0,Y 287.951,Z 543.154,A -85,B 0,C 180,E1 -17644.377,E2 -17644.377} C_VEL
LIN {X 0,Y 290.085,Z 530.53,A -85,B 0,C 180,E1 -17645.456,E2 -17645.456} C_VEL
LIN {X 0,Y 291.577,Z 519.29,A -85,B 0,C 180,E1 -17646.183,E2 -17646.183} C_VEL
LIN {X 0,Y 292.909,Z 505.328,A -85,B 0,C 180,E1 -17646.804,E2 -17646.804} C_VEL
LIN {X 0,Y 297.429,Z 444.935,A -85,B 0,C 180,E1 -17648.877,E2 -17648.877} C_VEL
LIN {X 0,Y 291.542,Z 431.827,A -85,B 0,C 180,E1 -17650.812,E2 -17650.812} C_VEL
LIN {X 0,Y 288.019,Z 425.371,A -85,B 0,C 180,E1 -17652.019,E2 -17652.019} C_VEL
LIN {X 0,Y 283.301,Z 417.776,A -85,B 0,C 180,E1 -17653.723,E2 -17653.723} C_VEL
LIN {X 0,Y 278.191,Z 410.259,A -85,B 0,C 180,E1 -17655.796,E2 -17655.796} C_VEL
LIN {X 0,Y 275.13,Z 406.086,A -85,B 0,C 180,E1 -17657.179,E2 -17657.179} C_VEL
LIN {X 0,Y 272.722,Z 403.014,A -85,B 0,C 180,E1 -17658.363,E2 -17658.363} C_VEL
LIN {X 0,Y 272.089,Z 401.708,A -85,B 0,C 180,E1 -17658.836,E2 -17658.836} C_VEL
LIN {X 0,Y 270.284,Z 397.913,A -85,B 0,C 180,E1 -17661.548,E2 -17661.548} C_VEL
LIN {X 0,Y 270.283,Z 397.816,A -85,B 0,C 180,E1 -17664.585,E2 -17664.585} C_VEL
LIN {X 0,Y 270.263,Z 397.819,A -85,B 0,C 180,E1 -17667.91,E2 -17667.91} C_VEL
LIN {X 0,Y 270.176,Z 397.83,A -85,B 0,C 180,E1 -17671.349,E2 -17671.349} C_VEL
LIN {X 0,Y 270.206,Z 397.826,A -85,B 0,C 180,E1 -17674.905,E2 -17674.905} C_VEL
LIN {X 0,Y 270.214,Z 397.824,A -85,B 0,C 180,E1 -17678.718,E2 -17678.718} C_VEL
LIN {X 0,Y 270.185,Z 397.828,A -85,B 0,C 180,E1 -17682.556,E2 -17682.556} C_VEL
LIN {X 0,Y 270.161,Z 397.877,A -85,B 0,C 180,E1 -17686.096,E2 -17686.096} C_VEL
LIN {X 0,Y 271.208,Z 400.741,A -85,B 0,C 180,E1 -17687.646,E2 -17687.646} C_VEL
LIN {X 0,Y 272.941,Z 403.202,A -85,B 0,C 180,E1 -17689.15,E2 -17689.15} C_VEL
LIN {X 0,Y 274.282,Z 405.67,A -85,B 0,C 180,E1 -17690.237,E2 -17690.237} C_VEL
LIN {X 0,Y 276.074,Z 407.915,A -85,B 0,C 180,E1 -17691.077,E2 -17691.077} C_VEL
LIN {X 0,Y 279.62,Z 412.724,A -85,B 0,C 180,E1 -17692.612,E2 -17692.612} C_VEL
LIN {X 0,Y 282.817,Z 417.371,A -85,B 0,C 180,E1 -17693.89,E2 -17693.89} C_VEL
LIN {X 0,Y 286.544,Z 423.182,A -85,B 0,C 180,E1 -17695.261,E2 -17695.261} C_VEL
LIN {X 0,Y 290.197,Z 432.226,A -85,B 0,C 180,E1 -17696.682,E2 -17696.682} C_VEL
LIN {X 0,Y 293.55,Z 441.635,A -85,B 0,C 180,E1 -17697.95,E2 -17697.95} C_VEL
LIN {X 0,Y 295.055,Z 453.797,A -85,B 0,C 180,E1 -17698.889,E2 -17698.889} C_VEL
LIN {X 0,Y 295.823,Z 464.143,A -85,B 0,C 180,E1 -17699.567,E2 -17699.567} C_VEL
LIN {X 0,Y 291.196,Z 525.056,A -85,B 0,C 180,E1 -17701.731,E2 -17701.731} C_VEL
LIN {X 0,Y 289.447,Z 538.31,A -85,B 0,C 180,E1 -17702.431,E2 -17702.431} C_VEL
LIN {X 0,Y 287.391,Z 550.132,A -85,B 0,C 180,E1 -17703.3,E2 -17703.3} C_VEL
LIN {X 0,Y 284.851,Z 563.214,A -85,B 0,C 180,E1 -17704.618,E2 -17704.618} C_VEL
LIN {X 0,Y 282.397,Z 573.711,A -85,B 0,C 180,E1 -17705.953,E2 -17705.953} C_VEL
LIN {X 0,Y 279.387,Z 585.29,A -85,B 0,C 180,E1 -17707.834,E2 -17707.834} C_VEL
LIN {X 0,Y 277.077,Z 593.833,A -85,B 0,C 180,E1 -17709.591,E2 -17709.591} C_VEL
LIN {X 0,Y 274.654,Z 602.212,A -85,B 0,C 180,E1 -17711.734,E2 -17711.734} C_VEL
LIN {X 0,Y 272.712,Z 609.039,A -85,B 0,C 180,E1 -17713.919,E2 -17713.919} C_VEL
LIN {X 0,Y 270.686,Z 615.331,A -85,B 0,C 180,E1 -17716.489,E2 -17716.489} C_VEL
LIN {X 0,Y 269.584,Z 619.417,A -85,B 0,C 180,E1 -17718.727,E2 -17718.727} C_VEL
LIN {X 0,Y 268.813,Z 622.47,A -85,B 0,C 180,E1 -17720.977,E2 -17720.977} C_VEL
LIN {X 0,Y 268.481,Z 623.93,A -85,B 0,C 180,E1 -17722.481,E2 -17722.481} C_VEL
LIN {X 0,Y 268.208,Z 625.337,A -85,B 0,C 180,E1 -17724.707,E2 -17724.707} C_VEL
LIN {X 0,Y 268.182,Z 625.826,A -85,B 0,C 180,E1 -17726.998,E2 -17726.998} C_VEL
LIN {X 0,Y 268.191,Z 626.793,A -85,B 0,C 180,E1 -17728.5,E2 -17728.5} C_VEL
LIN {X 0,Y 268.201,Z 627.375,A -85,B 0,C 180,E1 -17730.002,E2 -17730.002} C_VEL
LIN {X 0,Y 268.181,Z 627.546,A -85,B 0,C 180,E1 -17731.504,E2 -17731.504} C_VEL
LIN {X 0,Y 268.156,Z 627.274,A -85,B 0,C 180,E1 -17733.007,E2 -17733.007} C_VEL
LIN {X 0,Y 268.226,Z 625.55,A -85,B 0,C 180,E1 -17736.018,E2 -17736.018} C_VEL
LIN {X 0,Y 268.427,Z 624.079,A -85,B 0,C 180,E1 -17737.524,E2 -17737.524} C_VEL
LIN {X 0,Y 268.977,Z 621.04,A -85,B 0,C 180,E1 -17739.78,E2 -17739.78} C_VEL
LIN {X 0,Y 269.838,Z 616.955,A -85,B 0,C 180,E1 -17742.028,E2 -17742.028} C_VEL
LIN {X 0,Y 271.038,Z 611.74,A -85,B 0,C 180,E1 -17744.263,E2 -17744.263} C_VEL
LIN {X 0,Y 272.763,Z 605.199,A -85,B 0,C 180,E1 -17746.467,E2 -17746.467} C_VEL
LIN {X 0,Y 274.605,Z 597.123,A -85,B 0,C 180,E1 -17748.654,E2 -17748.654} C_VEL
LIN {X 0,Y 276.526,Z 588.869,A -85,B 0,C 180,E1 -17750.456,E2 -17750.456} C_VEL
LIN {X 0,Y 278.832,Z 578.859,A -85,B 0,C 180,E1 -17752.216,E2 -17752.216} C_VEL
LIN {X 0,Y 281.117,Z 567.598,A -85,B 0,C 180,E1 -17753.776,E2 -17753.776} C_VEL
LIN {X 0,Y 282.988,Z 556.66,A -85,B 0,C 180,E1 -17754.975,E2 -17754.975} C_VEL
LIN {X 0,Y 284.835,Z 544.638,A -85,B 0,C 180,E1 -17755.976,E2 -17755.976} C_VEL
LIN {X 0,Y 286.361,Z 532.34,A -85,B 0,C 180,E1 -17756.709,E2 -17756.709} C_VEL
LIN {X 0,Y 287.35,Z 518.859,A -85,B 0,C 180,E1 -17757.248,E2 -17757.248} C_VEL
LIN {X 0,Y 289.59,Z 462.204,A -85,B 0,C 180,E1 -17758.83,E2 -17758.83} C_VEL
LIN {X 0,Y 287.165,Z 445.46,A -85,B 0,C 180,E1 -17759.732,E2 -17759.732} C_VEL
LIN {X 0,Y 285.597,Z 437.654,A -85,B 0,C 180,E1 -17760.223,E2 -17760.223} C_VEL
LIN {X 0,Y 280.294,Z 425.9,A -85,B 0,C 180,E1 -17761.449,E2 -17761.449} C_VEL
LIN {X 0,Y 276.002,Z 417.52,A -85,B 0,C 180,E1 -17762.458,E2 -17762.458} C_VEL
LIN {X 0,Y 274.382,Z 413.951,A -85,B 0,C 180,E1 -17762.918,E2 -17762.918} C_VEL
LIN {X 0,Y 272.507,Z 406.093,A -85,B 0,C 180,E1 -17766.384,E2 -17766.384} C_VEL
LIN {X 0,Y 271.043,Z 400.807,A -85,B 0,C 180,E1 -17768.933,E2 -17768.933} C_VEL
LIN {X 0,Y 270.18,Z 397.834,A -85,B 0,C 180,E1 -17770.567,E2 -17770.567} C_VEL
LIN {X 0,Y 270.158,Z 397.832,A -85,B 0,C 180,E1 -17774.621,E2 -17774.621} C_VEL
LIN {X 0,Y 270.175,Z 397.829,A -85,B 0,C 180,E1 -17778.973,E2 -17778.973} C_VEL
LIN {X 0,Y 270.223,Z 397.819,A -85,B 0,C 180,E1 -17783.26,E2 -17783.26} C_VEL
LIN {X 0,Y 270.209,Z 397.821,A -85,B 0,C 180,E1 -17786.893,E2 -17786.893} C_VEL
LIN {X 0,Y 270.234,Z 397.815,A -85,B 0,C 180,E1 -17790.387,E2 -17790.387} C_VEL
LIN {X 0,Y 270.268,Z 397.809,A -85,B 0,C 180,E1 -17793.764,E2 -17793.764} C_VEL
LIN {X 0,Y 270.239,Z 397.812,A -85,B 0,C 180,E1 -17797.039,E2 -17797.039} C_VEL
LIN {X 0,Y 270.309,Z 397.809,A -85,B 0,C 180,E1 -17800.245,E2 -17800.245} C_VEL
LIN {X 0,Y 270.41,Z 397.791,A -85,B 0,C 180,E1 -17804.936,E2 -17804.936} C_VEL
LIN {X 0,Y 270.449,Z 397.786,A -85,B 0,C 180,E1 -17809.519,E2 -17809.519} C_VEL
LIN {X 0,Y 270.619,Z 397.769,A -85,B 0,C 180,E1 -17812.539,E2 -17812.539} C_VEL
LIN {X 0,Y 270.793,Z 397.754,A -85,B 0,C 180,E1 -17818.513,E2 -17818.513} C_VEL
LIN {X 0,Y 270.793,Z 397.75,A -85,B 0,C 180,E1 -17821.487,E2 -17821.487} C_VEL
LIN {X 0,Y 270.619,Z 397.773,A -85,B 0,C 180,E1 -17827.461,E2 -17827.461} C_VEL
LIN {X 0,Y 270.449,Z 397.799,A -85,B 0,C 180,E1 -17830.481,E2 -17830.481} C_VEL
LIN {X 0,Y 270.411,Z 397.803,A -85,B 0,C 180,E1 -17835.064,E2 -17835.064} C_VEL
LIN {X 0,Y 270.421,Z 397.849,A -85,B 0,C 180,E1 -17835.79,E2 -17835.79} C_VEL
LIN {X 0,Y 271.871,Z 403.486,A -85,B 0,C 180,E1 -17838.755,E2 -17838.755} C_VEL
LIN {X 0,Y 274.142,Z 407.593,A -85,B 0,C 180,E1 -17839.322,E2 -17839.322} C_VEL
LIN {X 0,Y 281.356,Z 420.84,A -85,B 0,C 180,E1 -17841.01,E2 -17841.01} C_VEL
LIN {X 0,Y 287.011,Z 432.735,A -85,B 0,C 180,E1 -17842.285,E2 -17842.285} C_VEL
LIN {X 0,Y 290.514,Z 441.553,A -85,B 0,C 180,E1 -17843.077,E2 -17843.077} C_VEL
LIN {X 0,Y 287.439,Z 510.562,A -85,B 0,C 180,E1 -17845.005,E2 -17845.005} C_VEL
LIN {X 0,Y 286.304,Z 523.706,A -85,B 0,C 180,E1 -17845.638,E2 -17845.638} C_VEL
LIN {X 0,Y 284.854,Z 536.073,A -85,B 0,C 180,E1 -17846.511,E2 -17846.511} C_VEL
LIN {X 0,Y 283.003,Z 548.509,A -85,B 0,C 180,E1 -17847.717,E2 -17847.717} C_VEL
LIN {X 0,Y 280.941,Z 559.923,A -85,B 0,C 180,E1 -17849.145,E2 -17849.145} C_VEL
LIN {X 0,Y 278.756,Z 570.328,A -85,B 0,C 180,E1 -17850.8,E2 -17850.8} C_VEL
LIN {X 0,Y 276.728,Z 579.126,A -85,B 0,C 180,E1 -17852.546,E2 -17852.546} C_VEL
LIN {X 0,Y 274.637,Z 587.384,A -85,B 0,C 180,E1 -17854.569,E2 -17854.569} C_VEL
LIN {X 0,Y 272.628,Z 595.074,A -85,B 0,C 180,E1 -17856.949,E2 -17856.949} C_VEL
LIN {X 0,Y 271.32,Z 600.281,A -85,B 0,C 180,E1 -17859.003,E2 -17859.003} C_VEL
LIN {X 0,Y 270.203,Z 604.393,A -85,B 0,C 180,E1 -17861.034,E2 -17861.034} C_VEL
LIN {X 0,Y 269.389,Z 607.579,A -85,B 0,C 180,E1 -17863.071,E2 -17863.071} C_VEL
LIN {X 0,Y 268.754,Z 609.925,A -85,B 0,C 180,E1 -17865.083,E2 -17865.083} C_VEL
LIN {X 0,Y 268.278,Z 611.573,A -85,B 0,C 180,E1 -17867.182,E2 -17867.182} C_VEL
LIN {X 0,Y 267.922,Z 612.463,A -85,B 0,C 180,E1 -17869.528,E2 -17869.528} C_VEL
LIN {X 0,Y 267.801,Z 612.351,A -85,B 0,C 180,E1 -17871.935,E2 -17871.935} C_VEL
LIN {X 0,Y 267.943,Z 610.88,A -85,B 0,C 180,E1 -17874.755,E2 -17874.755} C_VEL
LIN {X 0,Y 268.201,Z 608.696,A -85,B 0,C 180,E1 -17876.986,E2 -17876.986} C_VEL
LIN {X 0,Y 268.793,Z 604.825,A -85,B 0,C 180,E1 -17879.637,E2 -17879.637} C_VEL
LIN {X 0,Y 269.431,Z 600.106,A -85,B 0,C 180,E1 -17881.995,E2 -17881.995} C_VEL
LIN {X 0,Y 270.467,Z 593.337,A -85,B 0,C 180,E1 -17884.568,E2 -17884.568} C_VEL
LIN {X 0,Y 271.644,Z 585.985,A -85,B 0,C 180,E1 -17886.76,E2 -17886.76} C_VEL
LIN {X 0,Y 273.114,Z 577.115,A -85,B 0,C 180,E1 -17888.882,E2 -17888.882} C_VEL
LIN {X 0,Y 274.485,Z 568.453,A -85,B 0,C 180,E1 -17890.556,E2 -17890.556} C_VEL
LIN {X 0,Y 275.971,Z 557.915,A -85,B 0,C 180,E1 -17892.204,E2 -17892.204} C_VEL
LIN {X 0,Y 277.473,Z 546.409,A -85,B 0,C 180,E1 -17893.632,E2 -17893.632} C_VEL
LIN {X 0,Y 278.719,Z 534.935,A -85,B 0,C 180,E1 -17894.739,E2 -17894.739} C_VEL
LIN {X 0,Y 279.839,Z 521.527,A -85,B 0,C 180,E1 -17895.685,E2 -17895.685} C_VEL
LIN {X 0,Y 280.711,Z 508.106,A -85,B 0,C 180,E1 -17896.316,E2 -17896.316} C_VEL
LIN {X 0,Y 282.981,Z 436.364,A -85,B 0,C 180,E1 -17898.29,E2 -17898.29} C_VEL
LIN {X 0,Y 281.543,Z 429.8,A -85,B 0,C 180,E1 -17898.606,E2 -17898.606} C_VEL
LIN {X 0,Y 274.961,Z 411.607,A -85,B 0,C 180,E1 -17899.733,E2 -17899.733} C_VEL
LIN {X 0,Y 271.229,Z 401.554,A -85,B 0,C 180,E1 -17900.424,E2 -17900.424} C_VEL
LIN {X 0,Y 270.542,Z 397.787,A -85,B 0,C 180,E1 -17901.979,E2 -17901.979} C_VEL
LIN {X 0,Y 270.632,Z 397.774,A -85,B 0,C 180,E1 -17907.021,E2 -17907.021} C_VEL
LIN {X 0,Y 270.845,Z 397.747,A -85,B 0,C 180,E1 -17909.998,E2 -17909.998} C_VEL
LIN {X 0,Y 270.635,Z 397.769,A -85,B 0,C 180,E1 -17912.975,E2 -17912.975} C_VEL
LIN {X 0,Y 270.614,Z 397.772,A -85,B 0,C 180,E1 -17917.459,E2 -17917.459} C_VEL
LIN {X 0,Y 270.443,Z 397.798,A -85,B 0,C 180,E1 -17920.479,E2 -17920.479} C_VEL
LIN {X 0,Y 270.403,Z 397.801,A -85,B 0,C 180,E1 -17925.062,E2 -17925.062} C_VEL
LIN {X 0,Y 270.3,Z 397.81,A -85,B 0,C 180,E1 -17929.753,E2 -17929.753} C_VEL
LIN {X 0,Y 270.272,Z 397.815,A -85,B 0,C 180,E1 -17934.583,E2 -17934.583} C_VEL
LIN {X 0,Y 270.268,Z 397.812,A -85,B 0,C 180,E1 -17937.907,E2 -17937.907} C_VEL
LIN {X 0,Y 270.182,Z 397.828,A -85,B 0,C 180,E1 -17941.346,E2 -17941.346} C_VEL
LIN {X 0,Y 270.221,Z 397.823,A -85,B 0,C 180,E1 -17944.9,E2 -17944.9} C_VEL
LIN {X 0,Y 270.217,Z 397.824,A -85,B 0,C 180,E1 -17948.715,E2 -17948.715} C_VEL
LIN {X 0,Y 270.277,Z 397.818,A -85,B 0,C 180,E1 -17951.166,E2 -17951.166} C_VEL
LIN {X 0,Y 270.504,Z 399.125,A -85,B 0,C 180,E1 -17951.512,E2 -17951.512} C_VEL
LIN {X 0,Y 278.364,Z 424.654,A -85,B 0,C 180,E1 -17952.936,E2 -17952.936} C_VEL
LIN {X 0,Y 279.962,Z 435.142,A -85,B 0,C 180,E1 -17953.398,E2 -17953.398} C_VEL
LIN {X 0,Y 277.168,Z 509.203,A -85,B 0,C 180,E1 -17955.852,E2 -17955.852} C_VEL
LIN {X 0,Y 276.475,Z 522.013,A -85,B 0,C 180,E1 -17956.533,E2 -17956.533} C_VEL
LIN {X 0,Y 275.477,Z 535.488,A -85,B 0,C 180,E1 -17957.568,E2 -17957.568} C_VEL
LIN {X 0,Y 274.396,Z 547.049,A -85,B 0,C 180,E1 -17958.736,E2 -17958.736} C_VEL
LIN {X 0,Y 273.13,Z 559.381,A -85,B 0,C 180,E1 -17960.349,E2 -17960.349} C_VEL
LIN {X 0,Y 272.489,Z 565.072,A -85,B 0,C 180,E1 -17961.235,E2 -17961.235} C_VEL
LIN {X 0,Y 271.192,Z 569.602,A -85,B 0,C 180,E1 -17961.989,E2 -17961.989} C_VEL
LIN {X 0,Y 267.514,Z 576.54,A -85,B 0,C 180,E1 -17963.279,E2 -17963.279} C_VEL
LIN {X 0,Y 263.994,Z 582.963,A -85,B 0,C 180,E1 -17964.72,E2 -17964.72} C_VEL
LIN {X 0,Y 262.96,Z 586.662,A -85,B 0,C 180,E1 -17965.695,E2 -17965.695} C_VEL
LIN {X 0,Y 262.121,Z 594.173,A -85,B 0,C 180,E1 -17968.025,E2 -17968.025} C_VEL
LIN {X 0,Y 261.582,Z 599.75,A -85,B 0,C 180,E1 -17970.195,E2 -17970.195} C_VEL
LIN {X 0,Y 261.206,Z 604.88,A -85,B 0,C 180,E1 -17972.78,E2 -17972.78} C_VEL
LIN {X 0,Y 260.798,Z 608.544,A -85,B 0,C 180,E1 -17975.311,E2 -17975.311} C_VEL
LIN {X 0,Y 260.711,Z 610.971,A -85,B 0,C 180,E1 -17977.827,E2 -17977.827} C_VEL
LIN {X 0,Y 260.902,Z 612.303,A -85,B 0,C 180,E1 -17980.521,E2 -17980.521} C_VEL
LIN {X 0,Y 261.201,Z 612.411,A -85,B 0,C 180,E1 -17982.784,E2 -17982.784} C_VEL
LIN {X 0,Y 261.769,Z 611.575,A -85,B 0,C 180,E1 -17985.125,E2 -17985.125} C_VEL
LIN {X 0,Y 262.687,Z 609.605,A -85,B 0,C 180,E1 -17987.641,E2 -17987.641} C_VEL
LIN {X 0,Y 263.939,Z 606.487,A -85,B 0,C 180,E1 -17990.119,E2 -17990.119} C_VEL
LIN {X 0,Y 265.528,Z 602.479,A -85,B 0,C 180,E1 -17992.395,E2 -17992.395} C_VEL
LIN {X 0,Y 267.966,Z 595.685,A -85,B 0,C 180,E1 -17995.266,E2 -17995.266} C_VEL
LIN {X 0,Y 270.718,Z 587.754,A -85,B 0,C 180,E1 -17997.768,E2 -17997.768} C_VEL
LIN {X 0,Y 273.612,Z 578.682,A -85,B 0,C 180,E1 -18000,E2 -18000} C_VEL
LIN {X 0,Y 276.626,Z 568.209,A -85,B 0,C 180,E1 -18002.002,E2 -18002.002} C_VEL
LIN {X 0,Y 279.335,Z 557.72,A -85,B 0,C 180,E1 -18003.606,E2 -18003.606} C_VEL
LIN {X 0,Y 281.929,Z 546.022,A -85,B 0,C 180,E1 -18005.014,E2 -18005.014} C_VEL
LIN {X 0,Y 284.142,Z 534.162,A -85,B 0,C 180,E1 -18006.123,E2 -18006.123} C_VEL
LIN {X 0,Y 286.015,Z 521.335,A -85,B 0,C 180,E1 -18007.013,E2 -18007.013} C_VEL
LIN {X 0,Y 287.432,Z 508.396,A -85,B 0,C 180,E1 -18007.64,E2 -18007.64} C_VEL
LIN {X 0,Y 292.313,Z 447.574,A -85,B 0,C 180,E1 -18009.796,E2 -18009.796} C_VEL
LIN {X 0,Y 287.288,Z 436.121,A -85,B 0,C 180,E1 -18011.562,E2 -18011.562} C_VEL
LIN {X 0,Y 283.834,Z 429.783,A -85,B 0,C 180,E1 -18012.819,E2 -18012.819} C_VEL
LIN {X 0,Y 279.059,Z 421.968,A -85,B 0,C 180,E1 -18014.686,E2 -18014.686} C_VEL
LIN {X 0,Y 275.095,Z 415.894,A -85,B 0,C 180,E1 -18016.426,E2 -18016.426} C_VEL
LIN {X 0,Y 272.36,Z 412.134,A -85,B 0,C 180,E1 -18017.723,E2 -18017.723} C_VEL
LIN {X 0,Y 270.073,Z 408.986,A -85,B 0,C 180,E1 -18018.934,E2 -18018.934} C_VEL
LIN {X 0,Y 268.918,Z 407.545,A -85,B 0,C 180,E1 -18019.566,E2 -18019.566} C_VEL
LIN {X 0,Y 265.666,Z 403.461,A -85,B 0,C 180,E1 -18021.601,E2 -18021.601} C_VEL
LIN {X 0,Y 264.871,Z 402.404,A -85,B 0,C 180,E1 -18022.175,E2 -18022.175} C_VEL
LIN {X 0,Y 263.208,Z 398.698,A -85,B 0,C 180,E1 -18025.927,E2 -18025.927} C_VEL
LIN {X 0,Y 263.171,Z 398.704,A -85,B 0,C 180,E1 -18028.731,E2 -18028.731} C_VEL
LIN {X 0,Y 263.125,Z 398.709,A -85,B 0,C 180,E1 -18032.289,E2 -18032.289} C_VEL
LIN {X 0,Y 263.179,Z 398.702,A -85,B 0,C 180,E1 -18035.979,E2 -18035.979} C_VEL
LIN {X 0,Y 263.124,Z 398.711,A -85,B 0,C 180,E1 -18039.869,E2 -18039.869} C_VEL
LIN {X 0,Y 263.162,Z 398.837,A -85,B 0,C 180,E1 -18041.886,E2 -18041.886} C_VEL
LIN {X 0,Y 264.123,Z 401.56,A -85,B 0,C 180,E1 -18044.078,E2 -18044.078} C_VEL
LIN {X 0,Y 265.894,Z 403.864,A -85,B 0,C 180,E1 -18046.077,E2 -18046.077} C_VEL
LIN {X 0,Y 266.709,Z 405.554,A -85,B 0,C 180,E1 -18046.936,E2 -18046.936} C_VEL
LIN {X 0,Y 270.675,Z 410.551,A -85,B 0,C 180,E1 -18049.231,E2 -18049.231} C_VEL
LIN {X 0,Y 273.411,Z 414.131,A -85,B 0,C 180,E1 -18050.601,E2 -18050.601} C_VEL
LIN {X 0,Y 276.553,Z 418.502,A -85,B 0,C 180,E1 -18052.044,E2 -18052.044} C_VEL
LIN {X 0,Y 281.719,Z 426.282,A -85,B 0,C 180,E1 -18054.16,E2 -18054.16} C_VEL
LIN {X 0,Y 283.382,Z 429.697,A -85,B 0,C 180,E1 -18054.831,E2 -18054.831} C_VEL
LIN {X 0,Y 287.22,Z 439.793,A -85,B 0,C 180,E1 -18056.42,E2 -18056.42} C_VEL
LIN {X 0,Y 289.052,Z 445.55,A -85,B 0,C 180,E1 -18057.173,E2 -18057.173} C_VEL
LIN {X 0,Y 290.592,Z 462.112,A -85,B 0,C 180,E1 -18058.418,E2 -18058.418} C_VEL
LIN {X 0,Y 290.662,Z 466.471,A -85,B 0,C 180,E1 -18058.662,E2 -18058.662} C_VEL
LIN {X 0,Y 285.952,Z 524.283,A -85,B 0,C 180,E1 -18060.762,E2 -18060.762} C_VEL
LIN {X 0,Y 283.928,Z 538.842,A -85,B 0,C 180,E1 -18061.546,E2 -18061.546} C_VEL
LIN {X 0,Y 281.605,Z 551.358,A -85,B 0,C 180,E1 -18062.505,E2 -18062.505} C_VEL
LIN {X 0,Y 278.949,Z 564.131,A -85,B 0,C 180,E1 -18063.841,E2 -18063.841} C_VEL
LIN {X 0,Y 276.052,Z 575.449,A -85,B 0,C 180,E1 -18065.364,E2 -18065.364} C_VEL
LIN {X 0,Y 272.927,Z 586.584,A -85,B 0,C 180,E1 -18067.281,E2 -18067.281} C_VEL
LIN {X 0,Y 269.943,Z 596.646,A -85,B 0,C 180,E1 -18069.504,E2 -18069.504} C_VEL
LIN {X 0,Y 267.598,Z 604.229,A -85,B 0,C 180,E1 -18071.632,E2 -18071.632} C_VEL
LIN {X 0,Y 265.574,Z 610.571,A -85,B 0,C 180,E1 -18073.869,E2 -18073.869} C_VEL
LIN {X 0,Y 263.783,Z 615.683,A -85,B 0,C 180,E1 -18076.128,E2 -18076.128} C_VEL
LIN {X 0,Y 262.608,Z 619.635,A -85,B 0,C 180,E1 -18078.423,E2 -18078.423} C_VEL
LIN {X 0,Y 261.777,Z 622.545,A -85,B 0,C 180,E1 -18080.732,E2 -18080.732} C_VEL
LIN {X 0,Y 261.228,Z 624.932,A -85,B 0,C 180,E1 -18083.824,E2 -18083.824} C_VEL
LIN {X 0,Y 261.072,Z 625.473,A -85,B 0,C 180,E1 -18085.37,E2 -18085.37} C_VEL
LIN {X 0,Y 261.095,Z 625.593,A -85,B 0,C 180,E1 -18086.916,E2 -18086.916} C_VEL
LIN {X 0,Y 261.126,Z 627.134,A -85,B 0,C 180,E1 -18090.002,E2 -18090.002} C_VEL
LIN {X 0,Y 261.108,Z 627.341,A -85,B 0,C 180,E1 -18091.544,E2 -18091.544} C_VEL
LIN {X 0,Y 261.051,Z 627.108,A -85,B 0,C 180,E1 -18093.088,E2 -18093.088} C_VEL
LIN {X 0,Y 261.153,Z 625.433,A -85,B 0,C 180,E1 -18096.182,E2 -18096.182} C_VEL
LIN {X 0,Y 261.363,Z 624.005,A -85,B 0,C 180,E1 -18097.729,E2 -18097.729} C_VEL
LIN {X 0,Y 261.973,Z 621.019,A -85,B 0,C 180,E1 -18100.044,E2 -18100.044} C_VEL
LIN {X 0,Y 262.86,Z 617.004,A -85,B 0,C 180,E1 -18102.353,E2 -18102.353} C_VEL
LIN {X 0,Y 264.165,Z 611.862,A -85,B 0,C 180,E1 -18104.642,E2 -18104.642} C_VEL
LIN {X 0,Y 265.95,Z 605.419,A -85,B 0,C 180,E1 -18106.901,E2 -18106.901} C_VEL
LIN {X 0,Y 268.012,Z 596.929,A -85,B 0,C 180,E1 -18109.262,E2 -18109.262} C_VEL
LIN {X 0,Y 270.317,Z 587.481,A -85,B 0,C 180,E1 -18111.347,E2 -18111.347} C_VEL
LIN {X 0,Y 272.817,Z 577.154,A -85,B 0,C 180,E1 -18113.134,E2 -18113.134} C_VEL
LIN {X 0,Y 275.239,Z 565.607,A -85,B 0,C 180,E1 -18114.718,E2 -18114.718} C_VEL
LIN {X 0,Y 277.244,Z 554.279,A -85,B 0,C 180,E1 -18115.932,E2 -18115.932} C_VEL
LIN {X 0,Y 279.152,Z 541.453,A -85,B 0,C 180,E1 -18116.949,E2 -18116.949} C_VEL
LIN {X 0,Y 280.793,Z 527.932,A -85,B 0,C 180,E1 -18117.686,E2 -18117.686} C_VEL
LIN {X 0,Y 281.662,Z 512.984,A -85,B 0,C 180,E1 -18118.2,E2 -18118.2} C_VEL
LIN {X 0,Y 283.785,Z 463.631,A -85,B 0,C 180,E1 -18119.588,E2 -18119.588} C_VEL
LIN {X 0,Y 281.301,Z 446.251,A -85,B 0,C 180,E1 -18120.56,E2 -18120.56} C_VEL
LIN {X 0,Y 280.24,Z 440.95,A -85,B 0,C 180,E1 -18120.915,E2 -18120.915} C_VEL
LIN {X 0,Y 275.554,Z 430.267,A -85,B 0,C 180,E1 -18122.058,E2 -18122.058} C_VEL
LIN {X 0,Y 271.097,Z 421.502,A -85,B 0,C 180,E1 -18123.155,E2 -18123.155} C_VEL
LIN {X 0,Y 268.886,Z 417.358,A -85,B 0,C 180,E1 -18123.719,E2 -18123.719} C_VEL
LIN {X 0,Y 267.159,Z 413.806,A -85,B 0,C 180,E1 -18124.184,E2 -18124.184} C_VEL
LIN {X 0,Y 265.428,Z 406.67,A -85,B 0,C 180,E1 -18127.519,E2 -18127.519} C_VEL
LIN {X 0,Y 263.135,Z 398.713,A -85,B 0,C 180,E1 -18131.731,E2 -18131.731} C_VEL
LIN {X 0,Y 263.13,Z 398.711,A -85,B 0,C 180,E1 -18136.152,E2 -18136.152} C_VEL
LIN {X 0,Y 263.111,Z 398.704,A -85,B 0,C 180,E1 -18140.129,E2 -18140.129} C_VEL
LIN {X 0,Y 263.17,Z 398.702,A -85,B 0,C 180,E1 -18144.019,E2 -18144.019} C_VEL
LIN {X 0,Y 263.139,Z 398.707,A -85,B 0,C 180,E1 -18147.713,E2 -18147.713} C_VEL
LIN {X 0,Y 263.207,Z 398.698,A -85,B 0,C 180,E1 -18151.784,E2 -18151.784} C_VEL
LIN {X 0,Y 263.233,Z 398.696,A -85,B 0,C 180,E1 -18155.201,E2 -18155.201} C_VEL
LIN {X 0,Y 263.271,Z 398.691,A -85,B 0,C 180,E1 -18159.694,E2 -18159.694} C_VEL
LIN {X 0,Y 263.358,Z 398.672,A -85,B 0,C 180,E1 -18164.523,E2 -18164.523} C_VEL
LIN {X 0,Y 263.381,Z 398.666,A -85,B 0,C 180,E1 -18169.235,E2 -18169.235} C_VEL
LIN {X 0,Y 263.58,Z 398.647,A -85,B 0,C 180,E1 -18172.339,E2 -18172.339} C_VEL
LIN {X 0,Y 263.758,Z 398.629,A -85,B 0,C 180,E1 -18178.473,E2 -18178.473} C_VEL
LIN {X 0,Y 263.758,Z 398.627,A -85,B 0,C 180,E1 -18181.527,E2 -18181.527} C_VEL
LIN {X 0,Y 263.58,Z 398.651,A -85,B 0,C 180,E1 -18187.662,E2 -18187.662} C_VEL
LIN {X 0,Y 263.382,Z 398.68,A -85,B 0,C 180,E1 -18190.765,E2 -18190.765} C_VEL
LIN {X 0,Y 263.345,Z 398.786,A -85,B 0,C 180,E1 -18194.588,E2 -18194.588} C_VEL
LIN {X 0,Y 264.764,Z 403.966,A -85,B 0,C 180,E1 -18197.424,E2 -18197.424} C_VEL
LIN {X 0,Y 266.836,Z 407.583,A -85,B 0,C 180,E1 -18197.978,E2 -18197.978} C_VEL
LIN {X 0,Y 270.916,Z 414.621,A -85,B 0,C 180,E1 -18199.02,E2 -18199.02} C_VEL
LIN {X 0,Y 276.604,Z 425.252,A -85,B 0,C 180,E1 -18200.404,E2 -18200.404} C_VEL
LIN {X 0,Y 281.807,Z 436.327,A -85,B 0,C 180,E1 -18201.637,E2 -18201.637} C_VEL
LIN {X 0,Y 284.614,Z 443.244,A -85,B 0,C 180,E1 -18202.302,E2 -18202.302} C_VEL
LIN {X 0,Y 281.46,Z 511.084,A -85,B 0,C 180,E1 -18204.239,E2 -18204.239} C_VEL
LIN {X 0,Y 280.284,Z 524.222,A -85,B 0,C 180,E1 -18204.89,E2 -18204.89} C_VEL
LIN {X 0,Y 278.749,Z 536.556,A -85,B 0,C 180,E1 -18205.78,E2 -18205.78} C_VEL
LIN {X 0,Y 276.77,Z 549.179,A -85,B 0,C 180,E1 -18207.037,E2 -18207.037} C_VEL
LIN {X 0,Y 274.708,Z 559.991,A -85,B 0,C 180,E1 -18208.423,E2 -18208.423} C_VEL
LIN {X 0,Y 272.666,Z 569.325,A -85,B 0,C 180,E1 -18209.914,E2 -18209.914} C_VEL
LIN {X 0,Y 270.489,Z 578.431,A -85,B 0,C 180,E1 -18211.717,E2 -18211.717} C_VEL
LIN {X 0,Y 268.252,Z 586.843,A -85,B 0,C 180,E1 -18213.781,E2 -18213.781} C_VEL
LIN {X 0,Y 266.32,Z 593.79,A -85,B 0,C 180,E1 -18215.904,E2 -18215.904} C_VEL
LIN {X 0,Y 264.776,Z 599.384,A -85,B 0,C 180,E1 -18218.044,E2 -18218.044} C_VEL
LIN {X 0,Y 263.301,Z 604.676,A -85,B 0,C 180,E1 -18220.644,E2 -18220.644} C_VEL
LIN {X 0,Y 262.415,Z 607.922,A -85,B 0,C 180,E1 -18222.792,E2 -18222.792} C_VEL
LIN {X 0,Y 261.499,Z 610.935,A -85,B 0,C 180,E1 -18225.669,E2 -18225.669} C_VEL
LIN {X 0,Y 261.082,Z 612.17,A -85,B 0,C 180,E1 -18227.701,E2 -18227.701} C_VEL
LIN {X 0,Y 260.805,Z 612.699,A -85,B 0,C 180,E1 -18229.702,E2 -18229.702} C_VEL
LIN {X 0,Y 260.716,Z 612.593,A -85,B 0,C 180,E1 -18231.682,E2 -18231.682} C_VEL
LIN {X 0,Y 260.749,Z 611.612,A -85,B 0,C 180,E1 -18233.959,E2 -18233.959} C_VEL
LIN {X 0,Y 261.042,Z 609.395,A -85,B 0,C 180,E1 -18236.576,E2 -18236.576} C_VEL
LIN {X 0,Y 261.593,Z 605.711,A -85,B 0,C 180,E1 -18239.304,E2 -18239.304} C_VEL
LIN {X 0,Y 262.385,Z 600.347,A -85,B 0,C 180,E1 -18242.118,E2 -18242.118} C_VEL
LIN {X 0,Y 263.227,Z 594.948,A -85,B 0,C 180,E1 -18244.285,E2 -18244.285} C_VEL
LIN {X 0,Y 264.377,Z 588.088,A -85,B 0,C 180,E1 -18246.498,E2 -18246.498} C_VEL
LIN {X 0,Y 265.776,Z 579.623,A -85,B 0,C 180,E1 -18248.677,E2 -18248.677} C_VEL
LIN {X 0,Y 267.252,Z 570.721,A -85,B 0,C 180,E1 -18250.531,E2 -18250.531} C_VEL
LIN {X 0,Y 268.903,Z 560.143,A -85,B 0,C 180,E1 -18252.31,E2 -18252.31} C_VEL
LIN {X 0,Y 270.444,Z 548.57,A -85,B 0,C 180,E1 -18253.839,E2 -18253.839} C_VEL
LIN {X 0,Y 271.874,Z 536.1,A -85,B 0,C 180,E1 -18255.113,E2 -18255.113} C_VEL
LIN {X 0,Y 272.997,Z 523.924,A -85,B 0,C 180,E1 -18256.032,E2 -18256.032} C_VEL
LIN {X 0,Y 273.887,Z 510.499,A -85,B 0,C 180,E1 -18256.725,E2 -18256.725} C_VEL
LIN {X 0,Y 275.079,Z 477.356,A -85,B 0,C 180,E1 -18257.695,E2 -18257.695} C_VEL
LIN {X 0,Y 276.396,Z 437.246,A -85,B 0,C 180,E1 -18258.812,E2 -18258.812} C_VEL
LIN {X 0,Y 274.963,Z 431.24,A -85,B 0,C 180,E1 -18259.122,E2 -18259.122} C_VEL
LIN {X 0,Y 265.223,Z 404.792,A -85,B 0,C 180,E1 -18260.85,E2 -18260.85} C_VEL
LIN {X 0,Y 264.103,Z 401.742,A -85,B 0,C 180,E1 -18261.1,E2 -18261.1} C_VEL
LIN {X 0,Y 263.537,Z 398.658,A -85,B 0,C 180,E1 -18262.432,E2 -18262.432} C_VEL
LIN {X 0,Y 263.754,Z 398.633,A -85,B 0,C 180,E1 -18268.471,E2 -18268.471} C_VEL
LIN {X 0,Y 263.755,Z 398.631,A -85,B 0,C 180,E1 -18271.525,E2 -18271.525} C_VEL
LIN {X 0,Y 263.575,Z 398.649,A -85,B 0,C 180,E1 -18277.659,E2 -18277.659} C_VEL
LIN {X 0,Y 263.375,Z 398.677,A -85,B 0,C 180,E1 -18280.763,E2 -18280.763} C_VEL
LIN {X 0,Y 263.351,Z 398.681,A -85,B 0,C 180,E1 -18285.476,E2 -18285.476} C_VEL
LIN {X 0,Y 263.262,Z 398.69,A -85,B 0,C 180,E1 -18290.304,E2 -18290.304} C_VEL
LIN {X 0,Y 263.207,Z 398.696,A -85,B 0,C 180,E1 -18295.289,E2 -18295.289} C_VEL
LIN {X 0,Y 263.164,Z 398.696,A -85,B 0,C 180,E1 -18298.729,E2 -18298.729} C_VEL
LIN {X 0,Y 263.131,Z 398.707,A -85,B 0,C 180,E1 -18302.286,E2 -18302.286} C_VEL
LIN {X 0,Y 263.188,Z 398.701,A -85,B 0,C 180,E1 -18305.975,E2 -18305.975} C_VEL
LIN {X 0,Y 263.164,Z 398.704,A -85,B 0,C 180,E1 -18309.859,E2 -18309.859} C_VEL
LIN {X 0,Y 263.229,Z 398.791,A -85,B 0,C 180,E1 -18310.896,E2 -18310.896} C_VEL
LIN {X 0,Y 263.428,Z 399.701,A -85,B 0,C 180,E1 -18311.039,E2 -18311.039} C_VEL
LIN {X 0,Y 271.669,Z 426.25,A -85,B 0,C 180,E1 -18312.58,E2 -18312.58} C_VEL
LIN {X 0,Y 273.142,Z 436.227,A -85,B 0,C 180,E1 -18313.029,E2 -18313.029} C_VEL
LIN {X 0,Y 270.186,Z 510.332,A -85,B 0,C 180,E1 -18315.566,E2 -18315.566} C_VEL
LIN {X 0,Y 269.521,Z 522.552,A -85,B 0,C 180,E1 -18316.251,E2 -18316.251} C_VEL
LIN {X 0,Y 268.435,Z 536.439,A -85,B 0,C 180,E1 -18317.355,E2 -18317.355} C_VEL
LIN {X 0,Y 267.286,Z 548.593,A -85,B 0,C 180,E1 -18318.651,E2 -18318.651} C_VEL
LIN {X 0,Y 265.986,Z 560.467,A -85,B 0,C 180,E1 -18320.271,E2 -18320.271} C_VEL
LIN {X 0,Y 264.767,Z 571.248,A -85,B 0,C 180,E1 -18322.132,E2 -18322.132} C_VEL
LIN {X 0,Y 263.591,Z 580.411,A -85,B 0,C 180,E1 -18324.085,E2 -18324.085} C_VEL
LIN {X 0,Y 262.96,Z 586.662,A -85,B 0,C 180,E1 -18325.695,E2 -18325.695} C_VEL
LIN {X 0,Y 261.943,Z 590.172,A -85,B 0,C 180,E1 -18326.707,E2 -18326.707} C_VEL
LIN {X 0,Y 258.559,Z 595.359,A -85,B 0,C 180,E1 -18328.412,E2 -18328.412} C_VEL
LIN {X 0,Y 255.215,Z 599.887,A -85,B 0,C 180,E1 -18330.246,E2 -18330.246} C_VEL
LIN {X 0,Y 254.287,Z 602.366,A -85,B 0,C 180,E1 -18331.442,E2 -18331.442} C_VEL
LIN {X 0,Y 253.922,Z 606.353,A -85,B 0,C 180,E1 -18333.714,E2 -18333.714} C_VEL
LIN {X 0,Y 253.658,Z 609.412,A -85,B 0,C 180,E1 -18336.103,E2 -18336.103} C_VEL
LIN {X 0,Y 253.621,Z 611.669,A -85,B 0,C 180,E1 -18338.885,E2 -18338.885} C_VEL
LIN {X 0,Y 253.82,Z 612.419,A -85,B 0,C 180,E1 -18340.593,E2 -18340.593} C_VEL
LIN {X 0,Y 254.015,Z 612.683,A -85,B 0,C 180,E1 -18342.281,E2 -18342.281} C_VEL
LIN {X 0,Y 254.639,Z 612.089,A -85,B 0,C 180,E1 -18345.006,E2 -18345.006} C_VEL
LIN {X 0,Y 255.423,Z 610.659,A -85,B 0,C 180,E1 -18347.284,E2 -18347.284} C_VEL
LIN {X 0,Y 256.828,Z 607.616,A -85,B 0,C 180,E1 -18350.091,E2 -18350.091} C_VEL
LIN {X 0,Y 258.852,Z 602.95,A -85,B 0,C 180,E1 -18352.982,E2 -18352.982} C_VEL
LIN {X 0,Y 261.178,Z 597.063,A -85,B 0,C 180,E1 -18355.598,E2 -18355.598} C_VEL
LIN {X 0,Y 263.946,Z 589.716,A -85,B 0,C 180,E1 -18358.093,E2 -18358.093} C_VEL
LIN {X 0,Y 267.061,Z 580.659,A -85,B 0,C 180,E1 -18360.467,E2 -18360.467} C_VEL
LIN {X 0,Y 269.815,Z 572.174,A -85,B 0,C 180,E1 -18362.239,E2 -18362.239} C_VEL
LIN {X 0,Y 272.577,Z 562.507,A -85,B 0,C 180,E1 -18363.881,E2 -18363.881} C_VEL
LIN {X 0,Y 275.452,Z 551.067,A -85,B 0,C 180,E1 -18365.413,E2 -18365.413} C_VEL
LIN {X 0,Y 277.669,Z 540.523,A -85,B 0,C 180,E1 -18366.54,E2 -18366.54} C_VEL
LIN {X 0,Y 279.859,Z 528.067,A -85,B 0,C 180,E1 -18367.576,E2 -18367.576} C_VEL
LIN {X 0,Y 281.74,Z 514.457,A -85,B 0,C 180,E1 -18368.382,E2 -18368.382} C_VEL
LIN {X 0,Y 284.009,Z 489.2,A -85,B 0,C 180,E1 -18369.328,E2 -18369.328} C_VEL
LIN {X 0,Y 287.288,Z 450.275,A -85,B 0,C 180,E1 -18370.744,E2 -18370.744} C_VEL
LIN {X 0,Y 283.073,Z 440.287,A -85,B 0,C 180,E1 -18372.367,E2 -18372.367} C_VEL
LIN {X 0,Y 279.018,Z 432.751,A -85,B 0,C 180,E1 -18373.962,E2 -18373.962} C_VEL
LIN {X 0,Y 273.63,Z 424.002,A -85,B 0,C 180,E1 -18376.304,E2 -18376.304} C_VEL
LIN {X 0,Y 269.963,Z 418.544,A -85,B 0,C 180,E1 -18378.124,E2 -18378.124} C_VEL
LIN {X 0,Y 267.402,Z 414.96,A -85,B 0,C 180,E1 -18379.535,E2 -18379.535} C_VEL
LIN {X 0,Y 263.403,Z 409.712,A -85,B 0,C 180,E1 -18382.14,E2 -18382.14} C_VEL
LIN {X 0,Y 259.145,Z 404.627,A -85,B 0,C 180,E1 -18385.835,E2 -18385.835} C_VEL
LIN {X 0,Y 257.496,Z 402.952,A -85,B 0,C 180,E1 -18387.964,E2 -18387.964} C_VEL
LIN {X 0,Y 256.651,Z 401.568,A -85,B 0,C 180,E1 -18391.914,E2 -18391.914} C_VEL
LIN {X 0,Y 256.635,Z 401.55,A -85,B 0,C 180,E1 -18395.106,E2 -18395.106} C_VEL
LIN {X 0,Y 257.021,Z 402.249,A -85,B 0,C 180,E1 -18397.539,E2 -18397.539} C_VEL
LIN {X 0,Y 258.973,Z 404.575,A -85,B 0,C 180,E1 -18401.748,E2 -18401.748} C_VEL
LIN {X 0,Y 261.559,Z 408.419,A -85,B 0,C 180,E1 -18404.316,E2 -18404.316} C_VEL
LIN {X 0,Y 263.61,Z 410.602,A -85,B 0,C 180,E1 -18405.849,E2 -18405.849} C_VEL
LIN {X 0,Y 266.395,Z 414.374,A -85,B 0,C 180,E1 -18407.704,E2 -18407.704} C_VEL
LIN {X 0,Y 270.657,Z 420.117,A -85,B 0,C 180,E1 -18410.057,E2 -18410.057} C_VEL
LIN {X 0,Y 273.606,Z 424.45,A -85,B 0,C 180,E1 -18411.497,E2 -18411.497} C_VEL
LIN {X 0,Y 278.364,Z 431.838,A -85,B 0,C 180,E1 -18413.564,E2 -18413.564} C_VEL
LIN {X 0,Y 279.688,Z 434.791,A -85,B 0,C 180,E1 -18414.153,E2 -18414.153} C_VEL
LIN {X 0,Y 283.148,Z 444.357,A -85,B 0,C 180,E1 -18415.691,E2 -18415.691} C_VEL
LIN {X 0,Y 284.479,Z 449.047,A -85,B 0,C 180,E1 -18416.309,E2 -18416.309} C_VEL
LIN {X 0,Y 285.743,Z 464.321,A -85,B 0,C 180,E1 -18417.484,E2 -18417.484} C_VEL
LIN {X 0,Y 285.64,Z 468.493,A -85,B 0,C 180,E1 -18417.697,E2 -18417.697} C_VEL
LIN {X 0,Y 280.725,Z 524.934,A -85,B 0,C 180,E1 -18419.8,E2 -18419.8} C_VEL
LIN {X 0,Y 278.706,Z 538.548,A -85,B 0,C 180,E1 -18420.549,E2 -18420.549} C_VEL
LIN {X 0,Y 276.275,Z 550.961,A -85,B 0,C 180,E1 -18421.515,E2 -18421.515} C_VEL
LIN {X 0,Y 273.465,Z 563.661,A -85,B 0,C 180,E1 -18422.862,E2 -18422.862} C_VEL
LIN {X 0,Y 270.389,Z 575.019,A -85,B 0,C 180,E1 -18424.4,E2 -18424.4} C_VEL
LIN {X 0,Y 267.684,Z 584.329,A -85,B 0,C 180,E1 -18425.989,E2 -18425.989} C_VEL
LIN {X 0,Y 264.938,Z 592.931,A -85,B 0,C 180,E1 -18427.792,E2 -18427.792} C_VEL
LIN {X 0,Y 262.196,Z 601.169,A -85,B 0,C 180,E1 -18429.959,E2 -18429.959} C_VEL
LIN {X 0,Y 259.884,Z 608.215,A -85,B 0,C 180,E1 -18432.29,E2 -18432.29} C_VEL
LIN {X 0,Y 257.512,Z 614.583,A -85,B 0,C 180,E1 -18434.975,E2 -18434.975} C_VEL
LIN {X 0,Y 256.051,Z 618.731,A -85,B 0,C 180,E1 -18437.318,E2 -18437.318} C_VEL
LIN {X 0,Y 255.322,Z 620.896,A -85,B 0,C 180,E1 -18438.893,E2 -18438.893} C_VEL
LIN {X 0,Y 254.76,Z 622.637,A -85,B 0,C 180,E1 -18440.475,E2 -18440.475} C_VEL
LIN {X 0,Y 254.359,Z 623.967,A -85,B 0,C 180,E1 -18442.061,E2 -18442.061} C_VEL
LIN {X 0,Y 254.021,Z 625.25,A -85,B 0,C 180,E1 -18444.883,E2 -18444.883} C_VEL
LIN {X 0,Y 254.011,Z 625.361,A -85,B 0,C 180,E1 -18446.83,E2 -18446.83} C_VEL
LIN {X 0,Y 254.054,Z 626.891,A -85,B 0,C 180,E1 -18450.002,E2 -18450.002} C_VEL
LIN {X 0,Y 254.014,Z 627.125,A -85,B 0,C 180,E1 -18451.587,E2 -18451.587} C_VEL
LIN {X 0,Y 253.95,Z 626.945,A -85,B 0,C 180,E1 -18453.175,E2 -18453.175} C_VEL
LIN {X 0,Y 253.991,Z 626.185,A -85,B 0,C 180,E1 -18455.041,E2 -18455.041} C_VEL
LIN {X 0,Y 254.32,Z 623.932,A -85,B 0,C 180,E1 -18457.944,E2 -18457.944} C_VEL
LIN {X 0,Y 254.945,Z 621.003,A -85,B 0,C 180,E1 -18460.324,E2 -18460.324} C_VEL
LIN {X 0,Y 255.891,Z 617.05,A -85,B 0,C 180,E1 -18462.694,E2 -18462.694} C_VEL
LIN {X 0,Y 257.309,Z 611.973,A -85,B 0,C 180,E1 -18465.041,E2 -18465.041} C_VEL
LIN {X 0,Y 259.156,Z 605.629,A -85,B 0,C 180,E1 -18467.358,E2 -18467.358} C_VEL
LIN {X 0,Y 261.208,Z 597.73,A -85,B 0,C 180,E1 -18469.661,E2 -18469.661} C_VEL
LIN {X 0,Y 263.749,Z 587.973,A -85,B 0,C 180,E1 -18471.906,E2 -18471.906} C_VEL
LIN {X 0,Y 266.356,Z 577.861,A -85,B 0,C 180,E1 -18473.729,E2 -18473.729} C_VEL
LIN {X 0,Y 268.853,Z 566.504,A -85,B 0,C 180,E1 -18475.346,E2 -18475.346} C_VEL
LIN {X 0,Y 270.933,Z 555.451,A -85,B 0,C 180,E1 -18476.583,E2 -18476.583} C_VEL
LIN {X 0,Y 272.938,Z 543.206,A -85,B 0,C 180,E1 -18477.614,E2 -18477.614} C_VEL
LIN {X 0,Y 274.698,Z 529.581,A -85,B 0,C 180,E1 -18478.407,E2 -18478.407} C_VEL
LIN {X 0,Y 275.647,Z 516.145,A -85,B 0,C 180,E1 -18478.925,E2 -18478.925} C_VEL
LIN {X 0,Y 277.983,Z 464.421,A -85,B 0,C 180,E1 -18480.418,E2 -18480.418} C_VEL
LIN {X 0,Y 275.6,Z 447.48,A -85,B 0,C 180,E1 -18481.412,E2 -18481.412} C_VEL
LIN {X 0,Y 274.827,Z 443.85,A -85,B 0,C 180,E1 -18481.673,E2 -18481.673} C_VEL
LIN {X 0,Y 270.001,Z 432.865,A -85,B 0,C 180,E1 -18482.906,E2 -18482.906} C_VEL
LIN {X 0,Y 264.669,Z 422.38,A -85,B 0,C 180,E1 -18484.313,E2 -18484.313} C_VEL
LIN {X 0,Y 261.709,Z 417.043,A -85,B 0,C 180,E1 -18485.118,E2 -18485.118} C_VEL
LIN {X 0,Y 259.938,Z 413.432,A -85,B 0,C 180,E1 -18485.668,E2 -18485.668} C_VEL
LIN {X 0,Y 258.099,Z 406.505,A -85,B 0,C 180,E1 -18489.167,E2 -18489.167} C_VEL
LIN {X 0,Y 256.07,Z 399.591,A -85,B 0,C 180,E1 -18493.087,E2 -18493.087} C_VEL
LIN {X 0,Y 256.067,Z 399.586,A -85,B 0,C 180,E1 -18496.674,E2 -18496.674} C_VEL
LIN {X 0,Y 256.078,Z 399.585,A -85,B 0,C 180,E1 -18500.859,E2 -18500.859} C_VEL
LIN {X 0,Y 256.137,Z 399.573,A -85,B 0,C 180,E1 -18502.869,E2 -18502.869} C_VEL
LIN {X 0,Y 256.074,Z 399.58,A -85,B 0,C 180,E1 -18506.708,E2 -18506.708} C_VEL
LIN {X 0,Y 256.12,Z 399.573,A -85,B 0,C 180,E1 -18510.401,E2 -18510.401} C_VEL
LIN {X 0,Y 256.195,Z 399.571,A -85,B 0,C 180,E1 -18514.862,E2 -18514.862} C_VEL
LIN {X 0,Y 256.174,Z 399.576,A -85,B 0,C 180,E1 -18519.106,E2 -18519.106} C_VEL
LIN {X 0,Y 256.307,Z 399.555,A -85,B 0,C 180,E1 -18524.086,E2 -18524.086} C_VEL
LIN {X 0,Y 256.317,Z 399.547,A -85,B 0,C 180,E1 -18528.934,E2 -18528.934} C_VEL
LIN {X 0,Y 256.548,Z 399.525,A -85,B 0,C 180,E1 -18532.127,E2 -18532.127} C_VEL
LIN {X 0,Y 256.721,Z 399.505,A -85,B 0,C 180,E1 -18538.431,E2 -18538.431} C_VEL
LIN {X 0,Y 256.721,Z 399.503,A -85,B 0,C 180,E1 -18541.569,E2 -18541.569} C_VEL
LIN {X 0,Y 256.548,Z 399.529,A -85,B 0,C 180,E1 -18547.873,E2 -18547.873} C_VEL
LIN {X 0,Y 256.318,Z 399.558,A -85,B 0,C 180,E1 -18551.066,E2 -18551.066} C_VEL
LIN {X 0,Y 256.291,Z 399.743,A -85,B 0,C 180,E1 -18553.277,E2 -18553.277} C_VEL
LIN {X 0,Y 257.57,Z 404.204,A -85,B 0,C 180,E1 -18555.929,E2 -18555.929} C_VEL
LIN {X 0,Y 259.864,Z 408.108,A -85,B 0,C 180,E1 -18556.597,E2 -18556.597} C_VEL
LIN {X 0,Y 264.246,Z 415.28,A -85,B 0,C 180,E1 -18557.79,E2 -18557.79} C_VEL
LIN {X 0,Y 271.469,Z 428.666,A -85,B 0,C 180,E1 -18559.667,E2 -18559.667} C_VEL
LIN {X 0,Y 277.558,Z 441.995,A -85,B 0,C 180,E1 -18561.175,E2 -18561.175} C_VEL
LIN {X 0,Y 278.842,Z 445.346,A -85,B 0,C 180,E1 -18561.5,E2 -18561.5} C_VEL
LIN {X 0,Y 275.605,Z 511.021,A -85,B 0,C 180,E1 -18563.418,E2 -18563.418} C_VEL
LIN {X 0,Y 274.332,Z 524.489,A -85,B 0,C 180,E1 -18564.093,E2 -18564.093} C_VEL
LIN {X 0,Y 272.749,Z 536.817,A -85,B 0,C 180,E1 -18565.001,E2 -18565.001} C_VEL
LIN {X 0,Y 270.858,Z 548.51,A -85,B 0,C 180,E1 -18566.174,E2 -18566.174} C_VEL
LIN {X 0,Y 268.792,Z 558.957,A -85,B 0,C 180,E1 -18567.508,E2 -18567.508} C_VEL
LIN {X 0,Y 266.569,Z 568.599,A -85,B 0,C 180,E1 -18569.035,E2 -18569.035} C_VEL
LIN {X 0,Y 264.319,Z 577.806,A -85,B 0,C 180,E1 -18570.854,E2 -18570.854} C_VEL
LIN {X 0,Y 261.901,Z 586.314,A -85,B 0,C 180,E1 -18572.94,E2 -18572.94} C_VEL
LIN {X 0,Y 259.864,Z 593.293,A -85,B 0,C 180,E1 -18575.083,E2 -18575.083} C_VEL
LIN {X 0,Y 257.842,Z 600.152,A -85,B 0,C 180,E1 -18577.769,E2 -18577.769} C_VEL
LIN {X 0,Y 256.206,Z 605.581,A -85,B 0,C 180,E1 -18580.622,E2 -18580.622} C_VEL
LIN {X 0,Y 255.022,Z 609.482,A -85,B 0,C 180,E1 -18583.548,E2 -18583.548} C_VEL
LIN {X 0,Y 254.264,Z 611.79,A -85,B 0,C 180,E1 -18586.287,E2 -18586.287} C_VEL
LIN {X 0,Y 253.891,Z 612.693,A -85,B 0,C 180,E1 -18588.365,E2 -18588.365} C_VEL
LIN {X 0,Y 253.634,Z 612.887,A -85,B 0,C 180,E1 -18590.883,E2 -18590.883} C_VEL
LIN {X 0,Y 253.634,Z 612.03,A -85,B 0,C 180,E1 -18593.473,E2 -18593.473} C_VEL
LIN {X 0,Y 253.907,Z 609.779,A -85,B 0,C 180,E1 -18596.384,E2 -18596.384} C_VEL
LIN {X 0,Y 254.408,Z 606.631,A -85,B 0,C 180,E1 -18598.912,E2 -18598.912} C_VEL
LIN {X 0,Y 254.933,Z 602.96,A -85,B 0,C 180,E1 -18601.077,E2 -18601.077} C_VEL
LIN {X 0,Y 255.747,Z 597.766,A -85,B 0,C 180,E1 -18603.475,E2 -18603.475} C_VEL
LIN {X 0,Y 256.832,Z 591.491,A -85,B 0,C 180,E1 -18605.764,E2 -18605.764} C_VEL
LIN {X 0,Y 258.228,Z 583.251,A -85,B 0,C 180,E1 -18608.148,E2 -18608.148} C_VEL
LIN {X 0,Y 259.754,Z 574.521,A -85,B 0,C 180,E1 -18610.177,E2 -18610.177} C_VEL
LIN {X 0,Y 261.375,Z 564.914,A -85,B 0,C 180,E1 -18611.986,E2 -18611.986} C_VEL
LIN {X 0,Y 262.937,Z 554.127,A -85,B 0,C 180,E1 -18613.61,E2 -18613.61} C_VEL
LIN {X 0,Y 264.602,Z 541.522,A -85,B 0,C 180,E1 -18615.088,E2 -18615.088} C_VEL
LIN {X 0,Y 265.801,Z 529.774,A -85,B 0,C 180,E1 -18616.134,E2 -18616.134} C_VEL
LIN {X 0,Y 266.89,Z 516.2,A -85,B 0,C 180,E1 -18616.989,E2 -18616.989} C_VEL
LIN {X 0,Y 267.596,Z 502.717,A -85,B 0,C 180,E1 -18617.522,E2 -18617.522} C_VEL
LIN {X 0,Y 269.805,Z 438.219,A -85,B 0,C 180,E1 -18619.36,E2 -18619.36} C_VEL
LIN {X 0,Y 268.358,Z 432.553,A -85,B 0,C 180,E1 -18619.668,E2 -18619.668} C_VEL
LIN {X 0,Y 257.788,Z 404.391,A -85,B 0,C 180,E1 -18621.596,E2 -18621.596} C_VEL
LIN {X 0,Y 256.944,Z 401.993,A -85,B 0,C 180,E1 -18621.791,E2 -18621.791} C_VEL
LIN {X 0,Y 256.481,Z 399.537,A -85,B 0,C 180,E1 -18622.915,E2 -18622.915} C_VEL
LIN {X 0,Y 256.717,Z 399.51,A -85,B 0,C 180,E1 -18628.429,E2 -18628.429} C_VEL
LIN {X 0,Y 256.718,Z 399.508,A -85,B 0,C 180,E1 -18631.567,E2 -18631.567} C_VEL
LIN {X 0,Y 256.542,Z 399.526,A -85,B 0,C 180,E1 -18637.871,E2 -18637.871} C_VEL
LIN {X 0,Y 256.311,Z 399.556,A -85,B 0,C 180,E1 -18641.064,E2 -18641.064} C_VEL
LIN {X 0,Y 256.301,Z 399.562,A -85,B 0,C 180,E1 -18645.913,E2 -18645.913} C_VEL
LIN {X 0,Y 256.164,Z 399.572,A -85,B 0,C 180,E1 -18650.893,E2 -18650.893} C_VEL
LIN {X 0,Y 256.186,Z 399.57,A -85,B 0,C 180,E1 -18655.136,E2 -18655.136} C_VEL
LIN {X 0,Y 256.101,Z 399.578,A -85,B 0,C 180,E1 -18659.599,E2 -18659.599} C_VEL
LIN {X 0,Y 256.082,Z 399.586,A -85,B 0,C 180,E1 -18663.288,E2 -18663.288} C_VEL
LIN {X 0,Y 256.137,Z 399.579,A -85,B 0,C 180,E1 -18667.277,E2 -18667.277} C_VEL
LIN {X 0,Y 256.153,Z 399.575,A -85,B 0,C 180,E1 -18670.51,E2 -18670.51} C_VEL
LIN {X 0,Y 265.046,Z 428.122,A -85,B 0,C 180,E1 -18672.22,E2 -18672.22} C_VEL
LIN {X 0,Y 266.299,Z 436.907,A -85,B 0,C 180,E1 -18672.629,E2 -18672.629} C_VEL
LIN {X 0,Y 263.332,Z 509.526,A -85,B 0,C 180,E1 -18675.19,E2 -18675.19} C_VEL
LIN {X 0,Y 262.627,Z 522.323,A -85,B 0,C 180,E1 -18675.911,E2 -18675.911} C_VEL
LIN {X 0,Y 261.51,Z 536.078,A -85,B 0,C 180,E1 -18677.027,E2 -18677.027} C_VEL
LIN {X 0,Y 260.297,Z 548.571,A -85,B 0,C 180,E1 -18678.385,E2 -18678.385} C_VEL
LIN {X 0,Y 258.941,Z 560.911,A -85,B 0,C 180,E1 -18680.117,E2 -18680.117} C_VEL
LIN {X 0,Y 257.785,Z 570.661,A -85,B 0,C 180,E1 -18681.837,E2 -18681.837} C_VEL
LIN {X 0,Y 256.558,Z 580.248,A -85,B 0,C 180,E1 -18683.917,E2 -18683.917} C_VEL
LIN {X 0,Y 255.73,Z 588.235,A -85,B 0,C 180,E1 -18686.046,E2 -18686.046} C_VEL
LIN {X 0,Y 254.912,Z 595.349,A -85,B 0,C 180,E1 -18688.41,E2 -18688.41} C_VEL
LIN {X 0,Y 254.367,Z 601.67,A -85,B 0,C 180,E1 -18691.085,E2 -18691.085} C_VEL
LIN {X 0,Y 254.287,Z 602.366,A -85,B 0,C 180,E1 -18691.442,E2 -18691.442} C_VEL
LIN {X 0,Y 253.38,Z 604.643,A -85,B 0,C 180,E1 -18692.661,E2 -18692.661} C_VEL
LIN {X 0,Y 250.199,Z 607.688,A -85,B 0,C 180,E1 -18694.687,E2 -18694.687} C_VEL
LIN {X 0,Y 247.637,Z 609.629,A -85,B 0,C 180,E1 -18696.373,E2 -18696.373} C_VEL
LIN {X 0,Y 246.582,Z 610.832,A -85,B 0,C 180,E1 -18697.7,E2 -18697.7} C_VEL
LIN {X 0,Y 246.514,Z 611.155,A -85,B 0,C 180,E1 -18698.151,E2 -18698.151} C_VEL
LIN {X 0,Y 246.641,Z 612.323,A -85,B 0,C 180,E1 -18700.1,E2 -18700.1} C_VEL
LIN {X 0,Y 246.852,Z 612.793,A -85,B 0,C 180,E1 -18701.749,E2 -18701.749} C_VEL
LIN {X 0,Y 247.499,Z 612.56,A -85,B 0,C 180,E1 -18704.889,E2 -18704.889} C_VEL
LIN {X 0,Y 248.16,Z 611.571,A -85,B 0,C 180,E1 -18706.905,E2 -18706.905} C_VEL
LIN {X 0,Y 249.717,Z 608.753,A -85,B 0,C 180,E1 -18710.061,E2 -18710.061} C_VEL
LIN {X 0,Y 251.589,Z 604.871,A -85,B 0,C 180,E1 -18712.778,E2 -18712.778} C_VEL
LIN {X 0,Y 253.822,Z 599.748,A -85,B 0,C 180,E1 -18715.378,E2 -18715.378} C_VEL
LIN {X 0,Y 256.702,Z 592.849,A -85,B 0,C 180,E1 -18718.039,E2 -18718.039} C_VEL
LIN {X 0,Y 259.627,Z 585.255,A -85,B 0,C 180,E1 -18720.299,E2 -18720.299} C_VEL
LIN {X 0,Y 262.603,Z 576.835,A -85,B 0,C 180,E1 -18722.301,E2 -18722.301} C_VEL
LIN {X 0,Y 265.783,Z 566.95,A -85,B 0,C 180,E1 -18724.17,E2 -18724.17} C_VEL
LIN {X 0,Y 268.744,Z 556.527,A -85,B 0,C 180,E1 -18725.751,E2 -18725.751} C_VEL
LIN {X 0,Y 271.423,Z 545.676,A -85,B 0,C 180,E1 -18727.065,E2 -18727.065} C_VEL
LIN {X 0,Y 273.915,Z 533.498,A -85,B 0,C 180,E1 -18728.205,E2 -18728.205} C_VEL
LIN {X 0,Y 275.938,Z 521.111,A -85,B 0,C 180,E1 -18729.067,E2 -18729.067} C_VEL
LIN {X 0,Y 277.464,Z 508.105,A -85,B 0,C 180,E1 -18729.707,E2 -18729.707} C_VEL
LIN {X 0,Y 282.486,Z 453.06,A -85,B 0,C 180,E1 -18731.74,E2 -18731.74} C_VEL
LIN {X 0,Y 279.109,Z 444.916,A -85,B 0,C 180,E1 -18733.119,E2 -18733.119} C_VEL
LIN {X 0,Y 274.82,Z 436.908,A -85,B 0,C 180,E1 -18734.934,E2 -18734.934} C_VEL
LIN {X 0,Y 270.161,Z 428.982,A -85,B 0,C 180,E1 -18737.145,E2 -18737.145} C_VEL
LIN {X 0,Y 267.268,Z 424.621,A -85,B 0,C 180,E1 -18738.69,E2 -18738.69} C_VEL
LIN {X 0,Y 264.401,Z 420.439,A -85,B 0,C 180,E1 -18740.415,E2 -18740.415} C_VEL
LIN {X 0,Y 261.32,Z 416.192,A -85,B 0,C 180,E1 -18742.587,E2 -18742.587} C_VEL
LIN {X 0,Y 257.042,Z 410.955,A -85,B 0,C 180,E1 -18746.598,E2 -18746.598} C_VEL
LIN {X 0,Y 254.972,Z 409.007,A -85,B 0,C 180,E1 -18749.745,E2 -18749.745} C_VEL
LIN {X 0,Y 254.071,Z 408.139,A -85,B 0,C 180,E1 -18752.643,E2 -18752.643} C_VEL
LIN {X 0,Y 254.152,Z 408.343,A -85,B 0,C 180,E1 -18755.744,E2 -18755.744} C_VEL
LIN {X 0,Y 255.578,Z 409.907,A -85,B 0,C 180,E1 -18759.232,E2 -18759.232} C_VEL
LIN {X 0,Y 257.249,Z 411.332,A -85,B 0,C 180,E1 -18761.417,E2 -18761.417} C_VEL
LIN {X 0,Y 259.715,Z 415.118,A -85,B 0,C 180,E1 -18763.996,E2 -18763.996} C_VEL
LIN {X 0,Y 261.576,Z 417.209,A -85,B 0,C 180,E1 -18765.474,E2 -18765.474} C_VEL
LIN {X 0,Y 264.102,Z 420.759,A -85,B 0,C 180,E1 -18767.239,E2 -18767.239} C_VEL
LIN {X 0,Y 267.963,Z 426.203,A -85,B 0,C 180,E1 -18769.517,E2 -18769.517} C_VEL
LIN {X 0,Y 270.834,Z 430.564,A -85,B 0,C 180,E1 -18770.989,E2 -18770.989} C_VEL
LIN {X 0,Y 275.024,Z 437.285,A -85,B 0,C 180,E1 -18772.923,E2 -18772.923} C_VEL
LIN {X 0,Y 277.029,Z 442.448,A -85,B 0,C 180,E1 -18773.904,E2 -18773.904} C_VEL
LIN {X 0,Y 279.998,Z 451.69,A -85,B 0,C 180,E1 -18775.327,E2 -18775.327} C_VEL
LIN {X 0,Y 281,Z 466.468,A -85,B 0,C 180,E1 -18776.506,E2 -18776.506} C_VEL
LIN {X 0,Y 280.434,Z 474.37,A -85,B 0,C 180,E1 -18776.839,E2 -18776.839} C_VEL
LIN {X 0,Y 275.826,Z 524.163,A -85,B 0,C 180,E1 -18778.727,E2 -18778.727} C_VEL
LIN {X 0,Y 273.607,Z 538.367,A -85,B 0,C 180,E1 -18779.518,E2 -18779.518} C_VEL
LIN {X 0,Y 270.649,Z 552.526,A -85,B 0,C 180,E1 -18780.653,E2 -18780.653} C_VEL
LIN {X 0,Y 267.702,Z 564.799,A -85,B 0,C 180,E1 -18782.015,E2 -18782.015} C_VEL
LIN {X 0,Y 264.512,Z 575.859,A -85,B 0,C 180,E1 -18783.576,E2 -18783.576} C_VEL
LIN {X 0,Y 261.335,Z 585.844,A -85,B 0,C 180,E1 -18785.367,E2 -18785.367} C_VEL
LIN {X 0,Y 257.976,Z 595.596,A -85,B 0,C 180,E1 -18787.582,E2 -18787.582} C_VEL
LIN {X 0,Y 255.089,Z 603.513,A -85,B 0,C 180,E1 -18789.858,E2 -18789.858} C_VEL
LIN {X 0,Y 252.814,Z 609.866,A -85,B 0,C 180,E1 -18792.197,E2 -18792.197} C_VEL
LIN {X 0,Y 250.687,Z 615.006,A -85,B 0,C 180,E1 -18794.556,E2 -18794.556} C_VEL
LIN {X 0,Y 249.122,Z 619.005,A -85,B 0,C 180,E1 -18796.959,E2 -18796.959} C_VEL
LIN {X 0,Y 248.345,Z 621.08,A -85,B 0,C 180,E1 -18798.577,E2 -18798.577} C_VEL
LIN {X 0,Y 247.731,Z 622.741,A -85,B 0,C 180,E1 -18800.202,E2 -18800.202} C_VEL
LIN {X 0,Y 247.306,Z 623.955,A -85,B 0,C 180,E1 -18801.833,E2 -18801.833} C_VEL
LIN {X 0,Y 247.071,Z 624.747,A -85,B 0,C 180,E1 -18803.469,E2 -18803.469} C_VEL
LIN {X 0,Y 246.921,Z 625.138,A -85,B 0,C 180,E1 -18805.104,E2 -18805.104} C_VEL
LIN {X 0,Y 246.909,Z 625.123,A -85,B 0,C 180,E1 -18806.739,E2 -18806.739} C_VEL
LIN {X 0,Y 246.983,Z 626.644,A -85,B 0,C 180,E1 -18810.002,E2 -18810.002} C_VEL
LIN {X 0,Y 246.921,Z 626.907,A -85,B 0,C 180,E1 -18811.633,E2 -18811.633} C_VEL
LIN {X 0,Y 246.854,Z 626.772,A -85,B 0,C 180,E1 -18813.266,E2 -18813.266} C_VEL
LIN {X 0,Y 246.883,Z 626.202,A -85,B 0,C 180,E1 -18814.901,E2 -18814.901} C_VEL
LIN {X 0,Y 247.274,Z 623.858,A -85,B 0,C 180,E1 -18818.172,E2 -18818.172} C_VEL
LIN {X 0,Y 247.924,Z 620.988,A -85,B 0,C 180,E1 -18820.62,E2 -18820.62} C_VEL
LIN {X 0,Y 248.933,Z 617.111,A -85,B 0,C 180,E1 -18823.055,E2 -18823.055} C_VEL
LIN {X 0,Y 250.462,Z 612.121,A -85,B 0,C 180,E1 -18825.462,E2 -18825.462} C_VEL
LIN {X 0,Y 252.383,Z 605.872,A -85,B 0,C 180,E1 -18827.839,E2 -18827.839} C_VEL
LIN {X 0,Y 254.427,Z 598.528,A -85,B 0,C 180,E1 -18830.086,E2 -18830.086} C_VEL
LIN {X 0,Y 256.727,Z 590.251,A -85,B 0,C 180,E1 -18832.114,E2 -18832.114} C_VEL
LIN {X 0,Y 259.343,Z 580.665,A -85,B 0,C 180,E1 -18833.986,E2 -18833.986} C_VEL
LIN {X 0,Y 261.905,Z 570.095,A -85,B 0,C 180,E1 -18835.641,E2 -18835.641} C_VEL
LIN {X 0,Y 264.363,Z 558.39,A -85,B 0,C 180,E1 -18837.084,E2 -18837.084} C_VEL
